// TIA Portal V19 export
FUNCTION_BLOCK "A0304_Navetta_FB"   // FB103, LAD
// stored: MemoryReserve 100, SetENOAutomatically false
   VAR_INPUT
      AreaInterface : "AreaInterface";
      ZSI : "udt_ZoneSafetyInterface";
      DSI_Feed_Testa : "udt_DeviceSafetyInterface";
      DSI_Feed_Coda : "udt_DeviceSafetyInterface";
      DSI_Valve : "udt_DeviceSafetyInterface";
      DataIn : Struct
         OP_Vai_A_Prelievo : Bool;
         OP_Vai_A_Deposito : Bool;
         OP_Prelievo : Bool;
         OP_Deposito : Bool;
         UnloadBenchCaricoMatPres1 : Bool;
         UnloadBenchCaricoMatPres2 : Bool;
         UnloadBenchScaricoMatPres1 : Bool;
         UnloadBenchScaricoMatPres2 : Bool;
         PalettoInternoCoda_LsRest : Bool;
         PalettoInternoCoda_LsWork : Bool;
         PalettoInternoTesta_LsRest : Bool;
         PalettoInternoTesta_LsWork : Bool;
         PalettoEsternoCoda_LsRest : Bool;
         PalettoEsternoCoda_LsWork : Bool;
         PalettoEsternoTesta_LsRest : Bool;
         PalettoEsternoTesta_LsWork : Bool;
      END_STRUCT;
      CIn : Struct
         Manager : Struct
            EnableStopDoorOpeningReq : Bool;
            EnableStopInPhase : Bool;
            EnableStopProgrammed : Bool;
            Control_ON : Bool;
            CanMoveFreely { ExternalAccessible := 'False'; ExternalVisible := 'False'; ExternalWritable := 'False'} : Bool;
            Phase : Struct
               VAI_A_PRELIEVO : Bool;
               PRELIEVO : Bool;
               VAI_A_DEPOSITO : Bool;
               DEPOSITO : Bool;
            END_STRUCT;
         END_STRUCT;
         Sostegno : Struct
            ReadyForDeposito : Bool;
         END_STRUCT;
         Sollevatori : Struct
            Testa : Struct
               InPosDeposito : Bool;
               ActualPos : LReal;
            END_STRUCT;
            Coda : Struct
               InPosDeposito : Bool;
               ActualPos : LReal;
            END_STRUCT;
         END_STRUCT;
         AirOk : Bool;
         CycleModeShortPiece : Bool;
      END_STRUCT;
      Config : Struct
         Navetta : Struct
            Testa : Struct
               Ax : "Positioning_DOL_Machine_Config";
               PalettiEsterni : "ValveMachine_Config";
               PalettiInterni : "ValveMachine_Config";
            END_STRUCT;
            Coda : Struct
               Ax : "Positioning_DOL_Machine_Config";
               PalettiEsterni : "ValveMachine_Config";
               PalettiInterni : "ValveMachine_Config";
            END_STRUCT;
            DelayMissingCondition { ExternalAccessible := 'False'; ExternalVisible := 'False'; ExternalWritable := 'False'} : Time := T#0MS;
         END_STRUCT;
      END_STRUCT;
   END_VAR
   VAR_OUTPUT
      MachineInterface : "MachineInterface";
      COut : Struct
         Testa : Struct
            Ax : "Positioning_DOL_Machine_COut";
            PalettiEsterni : "ValveMachine_COut";
            PalettiInterni : "ValveMachine_COut";
         END_STRUCT;
         Coda : Struct
            Ax : "Positioning_DOL_Machine_COut";
            PalettiEsterni : "ValveMachine_COut";
            PalettiInterni : "ValveMachine_COut";
         END_STRUCT;
         Cumulativo : Struct
            PalettiEsterni : "ValveMachine_COut";
            PalettiInterni : "ValveMachine_COut";
         END_STRUCT;
         ReadyToRecive : Bool;
      END_STRUCT;
      DataOut : Struct
         Testa : Struct
            PalettoEsterno : Struct
               SbloccaggioStelo : Bool;   // 0= Bloccato
               Rest : Bool;
               Work : Bool;
            END_STRUCT;
            PalettoInterno : Struct
               SbloccaggioStelo : Bool;   // 0= Bloccato
               Rest : Bool;
               Work : Bool;
            END_STRUCT;
         END_STRUCT;
         Coda : Struct
            PalettoEsterno : Struct
               SbloccaggioStelo : Bool;
               Rest : Bool;
               Work : Bool;
            END_STRUCT;
            PalettoInterno : Struct
               SbloccaggioStelo : Bool;
               Rest : Bool;
               Work : Bool;
            END_STRUCT;
         END_STRUCT;
      END_STRUCT;
   END_VAR
   VAR_IN_OUT
      Par : Struct
         Ax_Man : "Positioning_DOL_Machine_Par";
         Ax_Testa_Pers : "Positioning_DOL_Machine_Pers_Data";
         Ax_Coda_Pers : "Positioning_DOL_Machine_Pers_Data";
         Enc : Struct
            Testa : "PosFbk_RTN";
            Coda : "PosFbk_RTN";
         END_STRUCT;
      END_STRUCT;
      Par_Mach : Struct
         PosPrePrelievo : LReal;
         PosPrelievo : LReal;
         PosDeposito : LReal;
         ToleranceWindow : LReal;
      END_STRUCT;
   END_VAR
   VAR
      Alarm : Struct
         Testa : Struct
            Ax : "Positioning_DOL_Machine_Alr";
            Enc : "PosFbk_Encoder_Alr";
            PalettiEsterni : "ValveAlr";
            PalettiInterni : "ValveAlr";
         END_STRUCT;
         Coda : Struct
            Ax : "Positioning_DOL_Machine_Alr";
            Enc : "PosFbk_Encoder_Alr";
            PalettiEsterni : "ValveAlr";
            PalettiInterni : "ValveAlr";
         END_STRUCT;
         CheckBothShutMove : Bool;
      END_STRUCT;
      Warning : Struct
         Testa : Struct
            Ax { S7_SetPoint := 'True'} : "Positioning_DOL_Machine_Wng";
            PalettiEsterni : "ValveMachine_Wng";
            PalettiInterni : "ValveMachine_Wng";
         END_STRUCT;
         Coda : Struct
            Ax { S7_SetPoint := 'True'} : "Positioning_DOL_Machine_Wng";
            PalettiEsterni : "ValveMachine_Wng";
            PalettiInterni : "ValveMachine_Wng";
         END_STRUCT;
         MissingCnd : Struct
            OP_VAI_A_PRELIEVO : Bool;   // Mancanza comando arresto
            OP_PRELIEVO : Bool;   // Mancanza consenso lavoro
            OP_VAI_A_DEPOSITO : Bool;   // Mancanza consenso lavoro
            OP_DEPOSITO : Bool;   // Mancanza consenso lavoro
         END_STRUCT;
      END_STRUCT;
      HMI : Struct
         Selection : Struct
            Ax : Int;   // 0= BOTH ; 1= HEAD ; 2= TAIL
            PalettiEsterni : Int;   // 0= BOTH ; 1= HEAD ; 2= TAIL
            PalettiInterni : Int;   // 0= BOTH ; 1= HEAD ; 2= TAIL
         END_STRUCT;
         Testa : Struct
            PbPreset : Bool;
            PresetValue : LReal;
         END_STRUCT;
         Coda : Struct
            PbPreset : Bool;
            PresetValue : LReal;
         END_STRUCT;
      END_STRUCT;
      Sts : Struct
         OP_CanMoveFreely : Bool;
         OP_Vai_A_Prelievo_Cnd : Bool;
         OP_Prelievo_Cnd : Bool;
         OP_Vai_A_Deposito_Cnd : Bool;
         OP_Deposito_Cnd : Bool;
         Coda_PermessoDaSynchOk : Bool;
         Testa_PermessoDaSynchOk : Bool;
         OutOfWorkSpace : Bool;   // Navetta fuori ingombro con impilatore e sollevatore
         GenCndFwd : Bool;
         GenCndBkw : Bool;
         ReloadAirRequest : Bool;
         InPosPrelievo : Bool;
         InPosPrePrelievo : Bool;
         InPosDeposito : Bool;
      END_STRUCT;
      Ctrl : Struct
         Man : Struct
            OP_Vai_A_Prelievo : Bool;
            OP_Prelievo : Bool;
            OP_Vai_A_Deposito : Bool;
            OP_Deposito : Bool;
         END_STRUCT;
         Aut : Struct
            OP_Vai_A_Prelievo : Bool;
            OP_Prelievo : Bool;
            OP_Vai_A_Deposito : Bool;
            OP_Deposito : Bool;
         END_STRUCT;
         OP_Vai_A_Prelievo : Bool;
         OP_Prelievo : Bool;
         OP_Vai_A_Deposito : Bool;
         OP_Deposito : Bool;
         ReloadAir { S7_SetPoint := 'True'} : Bool;
      END_STRUCT;
      Ax_Testa { S7_SetPoint := 'True'} : "Positioning_DOL_Machine_FB";
      Ax_Coda { S7_SetPoint := 'True'} : "Positioning_DOL_Machine_FB";
      PalettiEsterni_Testa { S7_SetPoint := 'True'} : "ValveMachine_FB";
      PalettiEsterni_Coda { S7_SetPoint := 'True'} : "ValveMachine_FB";
      PalettiInterni_Testa { S7_SetPoint := 'True'} : "ValveMachine_FB";
      PalettiInterni_Coda { S7_SetPoint := 'True'} : "ValveMachine_FB";
      BloccaggioStelo_PalettoEsterno_Testa { S7_SetPoint := 'True'} : "Valve";
      BloccaggioStelo_PalettoEsterno_Coda { S7_SetPoint := 'True'} : "Valve";
      Enc_Testa : "PosFbk_SickAFM60";
      Enc_Testa_ITF : "PosFbk_ITF";
      Enc_Coda : "PosFbk_SickAFM60";
      Enc_Coda_ITF : "PosFbk_ITF";
      AUX { ExternalAccessible := 'False'; ExternalVisible := 'False'; ExternalWritable := 'False'} : Struct
         OP_Vai_A_Prelievo : Bool;
         OP_Prelievo : Bool;
         OP_Vai_A_Deposito : Bool;
         OP_Deposito : Bool;
         AirOk : Bool;
         Clock250 : Bool;
      END_STRUCT;
      TON_OP_VAI_A_PRELIEVO_MissingCnd : IEC_TIMER;
      TON_OP_PRELIEVO_MissingCnd : IEC_TIMER;
      TON_OP_VAI_A_DEPOSITO_MissingCnd : IEC_TIMER;
      TON_OP_DEPOSITO_MissingCnd : IEC_TIMER;
      TON_CheckShuttleMove { S7_SetPoint := 'True'} : IEC_TIMER;
      TON_ReloadAir { S7_SetPoint := 'True'} : IEC_TIMER;
      TON_CheckAxis { S7_SetPoint := 'True'} : IEC_TIMER;
      CheckAxisSynch { ExternalAccessible := 'False'; ExternalVisible := 'False'; ExternalWritable := 'False'} : "CheckAxisSynch";
      Sts_PosAxis { S7_SetPoint := 'True'} : Int;
   END_VAR
   VAR_TEMP
      PE : Struct
         OP_Vai_A_Prelievo : Bool;
         OP_Prelievo : Bool;
         OP_Vai_A_Deposito : Bool;
         OP_Deposito : Bool;
         Clock250 : Bool;
      END_STRUCT;
      NE : Struct
         AirOk : Bool;
      END_STRUCT;
      AxTesta_InPosDeposito : Bool;
      AxCoda_InPosDeposito : Bool;
      AxTesta_InPosPrelievo : Bool;
      AxCoda_InPosPrelievo : Bool;
      AxCoda_InPosPrePrelievo : Bool;
      AxTesta_InPosPrePrelievo : Bool;
   END_VAR
   VAR CONSTANT
      "Ax_Fuori Ingombro" : LReal := 800.0;
      MaxDistance : LReal := 5.0;
      MinDistance : LReal := 0.5;
   END_VAR
   // Config.Navetta.Testa.Ax.DelayMissingCondition := T#3S;
   // Config.Navetta.Testa.Ax.CyclicOBTime_ms := 10.0;
   // Config.Navetta.Testa.Ax.Ax.limitMinus := -25.0;
   // Config.Navetta.Testa.Ax.Ax.limitPlus := 2175.0;
   // Config.Navetta.Testa.Ax.Ax.Backlash := 0.0;
   // Config.Navetta.Testa.Ax.Ax.BacklashActivation := FALSE;
   // Config.Navetta.Testa.Ax.Ax.ToleranceWindow := 0.1;
   // Config.Navetta.Testa.Ax.Ax.ToleranceWindowDelay := T#100MS;
   // Config.Navetta.Testa.Ax.Ax.PreCutOff := 0.0;
   // Config.Navetta.Testa.Ax.Ax.PreEndLowSpeed := 0.0;
   // Config.Navetta.Testa.Ax.Ax.PreEndMedSpeed := 0.0;
   // Config.Navetta.Testa.Ax.Ax.ChangeDirectionDelay := T#0MS;
   // Config.Navetta.Testa.Ax.Ax.StandstillVelocity := 0.5;
   // Config.Navetta.Testa.Ax.Ax.StandStillDelay := T#100MS;
   // Config.Navetta.Testa.Ax.Ax.HomingDirection := FALSE;
   // Config.Navetta.Testa.Ax.Ax.RecallTime := 0.0;
   // Config.Navetta.Testa.Ax.Ax.VelocityFilter_T := 10.0;
   // Config.Navetta.Testa.Ax.Ax.VelocityMeasUnit := 2;
   // Config.Navetta.Testa.Ax.Ax.PosFbkDisabled := FALSE;
   // Config.Navetta.Testa.Ax.Ax.FbkCtrlDisabled := TRUE;
   // Config.Navetta.Testa.Ax.Ax_UM2."m" := 1.0;
   // Config.Navetta.Testa.Ax.Ax_UM2.q := 0.0;
   // Config.Navetta.Testa.Ax.S120.SpeedMotor.ReferenceVelocity := 2000.0;
   // Config.Navetta.Testa.Ax.S120.SpeedMotor.InvertDirection := FALSE;
   // Config.Navetta.Testa.Ax.S120.PowerOffDelay := T#5S;
   // Config.Navetta.Testa.Ax.S120.StandstillVelocity := 50.0;
   // Config.Navetta.Testa.Ax.S120.AccTime := 0.25;
   // Config.Navetta.Testa.Ax.S120.DecTime := 0.25;
   // Config.Navetta.Testa.Ax.Fan.Presence := FALSE;
   // Config.Navetta.Testa.Ax.Fan.DelayOff := T#10M;
   // Config.Navetta.Testa.Ax.Brake_Presence := FALSE;
   // Config.Navetta.Testa.PalettiEsterni.DelayPressureRunningTimeout := T#3S;
   // Config.Navetta.Testa.PalettiEsterni.DelayMissingCondition := T#3S;
   // Config.Navetta.Testa.PalettiEsterni.Rest_LsQty := 1;
   // Config.Navetta.Testa.PalettiEsterni.Work_LsQty := 1;
   // Config.Navetta.Testa.PalettiEsterni.Rest_RetainAut := FALSE;
   // Config.Navetta.Testa.PalettiEsterni.Work_RetainAut := FALSE;
   // Config.Navetta.Testa.PalettiEsterni.V.RestLimSwitchExist := TRUE;
   // Config.Navetta.Testa.PalettiEsterni.V.WorkLimSwitchExist := TRUE;
   // Config.Navetta.Testa.PalettiEsterni.V.CheckOilInPressure := FALSE;
   // Config.Navetta.Testa.PalettiEsterni.V.CutRestWhenIsAtRest := TRUE;
   // Config.Navetta.Testa.PalettiEsterni.V.CutWorkWhenIsAtWork := TRUE;
   // Config.Navetta.Testa.PalettiEsterni.V.RestTime := T#0MS;
   // Config.Navetta.Testa.PalettiEsterni.V.WorkTime := T#0MS;
   // Config.Navetta.Testa.PalettiEsterni.V.RestTimeOut := T#6S;
   // Config.Navetta.Testa.PalettiEsterni.V.WorkTimeOut := T#6S;
   // Config.Navetta.Testa.PalettiInterni.DelayPressureRunningTimeout := T#3S;
   // Config.Navetta.Testa.PalettiInterni.DelayMissingCondition := T#3S;
   // Config.Navetta.Testa.PalettiInterni.Rest_LsQty := 1;
   // Config.Navetta.Testa.PalettiInterni.Work_LsQty := 1;
   // Config.Navetta.Testa.PalettiInterni.Rest_RetainAut := FALSE;
   // Config.Navetta.Testa.PalettiInterni.Work_RetainAut := FALSE;
   // Config.Navetta.Testa.PalettiInterni.V.RestLimSwitchExist := TRUE;
   // Config.Navetta.Testa.PalettiInterni.V.WorkLimSwitchExist := TRUE;
   // Config.Navetta.Testa.PalettiInterni.V.CheckOilInPressure := FALSE;
   // Config.Navetta.Testa.PalettiInterni.V.CutRestWhenIsAtRest := TRUE;
   // Config.Navetta.Testa.PalettiInterni.V.CutWorkWhenIsAtWork := TRUE;
   // Config.Navetta.Testa.PalettiInterni.V.RestTime := T#0MS;
   // Config.Navetta.Testa.PalettiInterni.V.WorkTime := T#0MS;
   // Config.Navetta.Testa.PalettiInterni.V.RestTimeOut := T#6S;
   // Config.Navetta.Testa.PalettiInterni.V.WorkTimeOut := T#6S;
   // Config.Navetta.Coda.Ax.DelayMissingCondition := T#3S;
   // Config.Navetta.Coda.Ax.CyclicOBTime_ms := 10.0;
   // Config.Navetta.Coda.Ax.Ax.limitMinus := -25.0;
   // Config.Navetta.Coda.Ax.Ax.limitPlus := 2175.0;
   // Config.Navetta.Coda.Ax.Ax.Backlash := 0.0;
   // Config.Navetta.Coda.Ax.Ax.BacklashActivation := FALSE;
   // Config.Navetta.Coda.Ax.Ax.ToleranceWindow := 0.1;
   // Config.Navetta.Coda.Ax.Ax.ToleranceWindowDelay := T#100MS;
   // Config.Navetta.Coda.Ax.Ax.PreCutOff := 0.0;
   // Config.Navetta.Coda.Ax.Ax.PreEndLowSpeed := 0.0;
   // Config.Navetta.Coda.Ax.Ax.PreEndMedSpeed := 0.0;
   // Config.Navetta.Coda.Ax.Ax.ChangeDirectionDelay := T#0MS;
   // Config.Navetta.Coda.Ax.Ax.StandstillVelocity := 0.5;
   // Config.Navetta.Coda.Ax.Ax.StandStillDelay := T#100MS;
   // Config.Navetta.Coda.Ax.Ax.HomingDirection := FALSE;
   // Config.Navetta.Coda.Ax.Ax.RecallTime := 0.0;
   // Config.Navetta.Coda.Ax.Ax.VelocityFilter_T := 10.0;
   // Config.Navetta.Coda.Ax.Ax.VelocityMeasUnit := 2;
   // Config.Navetta.Coda.Ax.Ax.PosFbkDisabled := FALSE;
   // Config.Navetta.Coda.Ax.Ax.FbkCtrlDisabled := TRUE;
   // Config.Navetta.Coda.Ax.Ax_UM2."m" := 1.0;
   // Config.Navetta.Coda.Ax.Ax_UM2.q := 0.0;
   // Config.Navetta.Coda.Ax.S120.SpeedMotor.ReferenceVelocity := 2200.0;
   // Config.Navetta.Coda.Ax.S120.SpeedMotor.InvertDirection := FALSE;
   // Config.Navetta.Coda.Ax.S120.PowerOffDelay := T#5S;
   // Config.Navetta.Coda.Ax.S120.StandstillVelocity := 50.0;
   // Config.Navetta.Coda.Ax.S120.AccTime := 0.25;
   // Config.Navetta.Coda.Ax.S120.DecTime := 0.25;
   // Config.Navetta.Coda.Ax.Fan.Presence := FALSE;
   // Config.Navetta.Coda.Ax.Fan.DelayOff := T#10M;
   // Config.Navetta.Coda.Ax.Brake_Presence := FALSE;
   // Config.Navetta.Coda.PalettiEsterni.DelayPressureRunningTimeout := T#3S;
   // Config.Navetta.Coda.PalettiEsterni.DelayMissingCondition := T#3S;
   // Config.Navetta.Coda.PalettiEsterni.Rest_LsQty := 1;
   // Config.Navetta.Coda.PalettiEsterni.Work_LsQty := 1;
   // Config.Navetta.Coda.PalettiEsterni.Rest_RetainAut := FALSE;
   // Config.Navetta.Coda.PalettiEsterni.Work_RetainAut := FALSE;
   // Config.Navetta.Coda.PalettiEsterni.V.RestLimSwitchExist := TRUE;
   // Config.Navetta.Coda.PalettiEsterni.V.WorkLimSwitchExist := TRUE;
   // Config.Navetta.Coda.PalettiEsterni.V.CheckOilInPressure := FALSE;
   // Config.Navetta.Coda.PalettiEsterni.V.CutRestWhenIsAtRest := TRUE;
   // Config.Navetta.Coda.PalettiEsterni.V.CutWorkWhenIsAtWork := TRUE;
   // Config.Navetta.Coda.PalettiEsterni.V.RestTime := T#0MS;
   // Config.Navetta.Coda.PalettiEsterni.V.WorkTime := T#0MS;
   // Config.Navetta.Coda.PalettiEsterni.V.RestTimeOut := T#6S;
   // Config.Navetta.Coda.PalettiEsterni.V.WorkTimeOut := T#6S;
   // Config.Navetta.Coda.PalettiInterni.DelayPressureRunningTimeout := T#3S;
   // Config.Navetta.Coda.PalettiInterni.DelayMissingCondition := T#3S;
   // Config.Navetta.Coda.PalettiInterni.Rest_LsQty := 1;
   // Config.Navetta.Coda.PalettiInterni.Work_LsQty := 1;
   // Config.Navetta.Coda.PalettiInterni.Rest_RetainAut := FALSE;
   // Config.Navetta.Coda.PalettiInterni.Work_RetainAut := FALSE;
   // Config.Navetta.Coda.PalettiInterni.V.RestLimSwitchExist := TRUE;
   // Config.Navetta.Coda.PalettiInterni.V.WorkLimSwitchExist := TRUE;
   // Config.Navetta.Coda.PalettiInterni.V.CheckOilInPressure := FALSE;
   // Config.Navetta.Coda.PalettiInterni.V.CutRestWhenIsAtRest := TRUE;
   // Config.Navetta.Coda.PalettiInterni.V.CutWorkWhenIsAtWork := TRUE;
   // Config.Navetta.Coda.PalettiInterni.V.RestTime := T#0MS;
   // Config.Navetta.Coda.PalettiInterni.V.WorkTime := T#0MS;
   // Config.Navetta.Coda.PalettiInterni.V.RestTimeOut := T#6S;
   // Config.Navetta.Coda.PalettiInterni.V.WorkTimeOut := T#6S;
   VAR_TEMP   // added for the SCL form of the ladder/FBD networks
      _w1 : Bool;
      _w2 : Bool;
      _w3 : Bool;
      _w4 : Bool;
   END_VAR
BEGIN

REGION Network 1 (SCL): Reset allarmi
   IF #AreaInterface.RstAlarms THEN
       #Alarm.CheckBothShutMove := FALSE;
   END_IF;
END_REGION

REGION Network 2: <+>
END_REGION

REGION Network 3: <<<<<<<<<<<<<<<<<<< OPERAZIONI >>>>>>>>>>>>>>>>>>>>>>>>
END_REGION

REGION Network 4: Operazione può muoversi liberamente perchè non sposta nessun BEAM
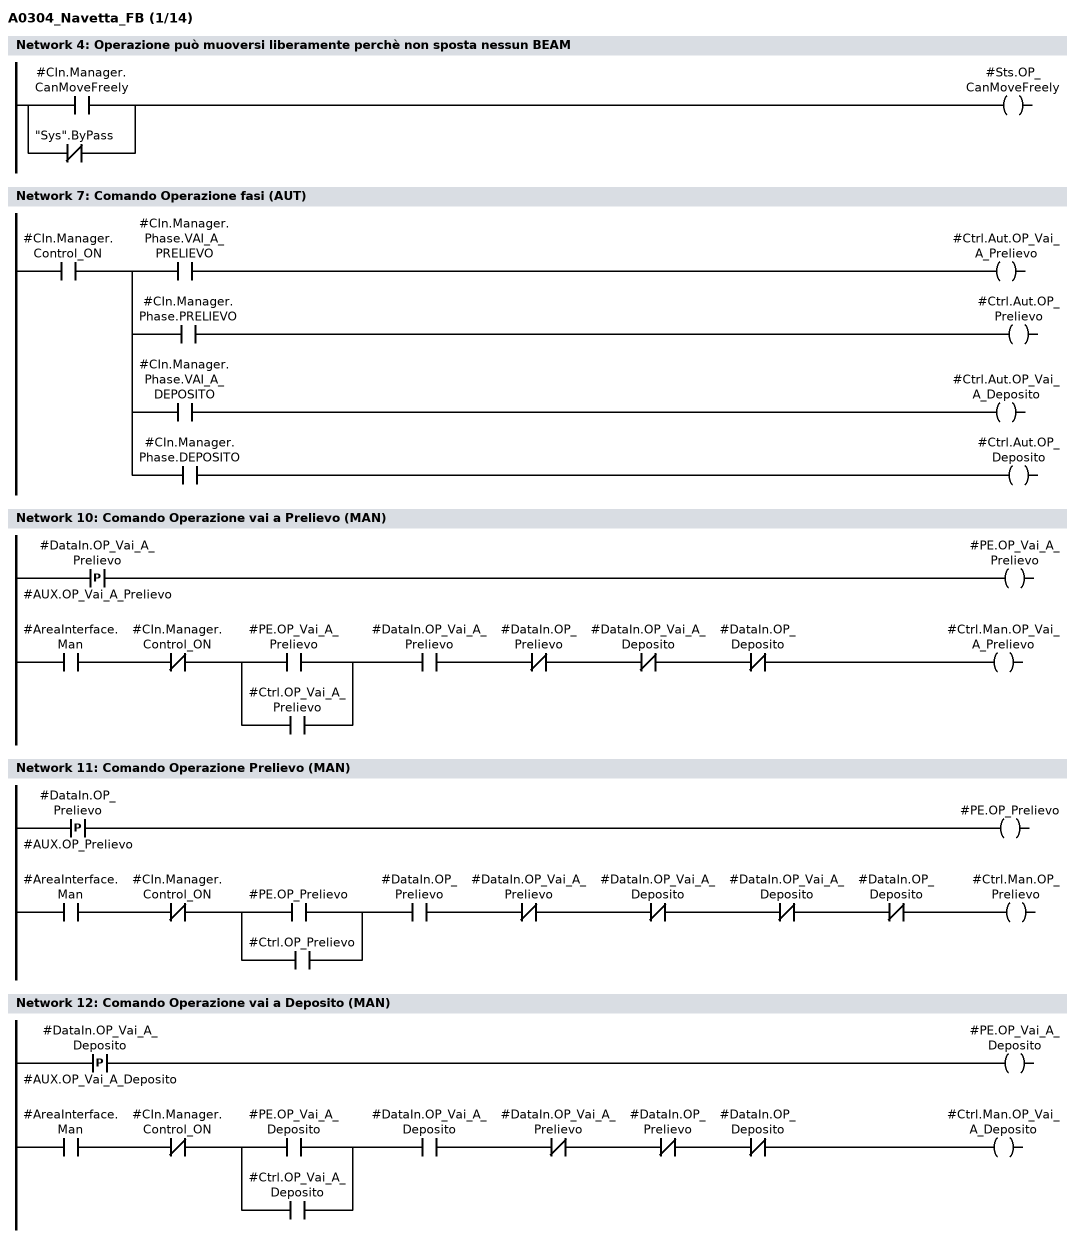
   RUNG wire#powerrail
      Contact( #CIn.Manager.CanMoveFreely )
      wire#w1
      Coil( #Sts.OP_CanMoveFreely )
   END_RUNG
   RUNG wire#powerrail
      I_Contact( "Sys".ByPass )
   END_RUNG wire#w1
   // the same network as SCL:
   #Sts.OP_CanMoveFreely := #CIn.Manager.CanMoveFreely OR NOT "Sys".ByPass;
END_REGION

REGION Network 5: <+>
END_REGION

REGION Network 6: < OPERAZIONI AUTOMATICO >
END_REGION

REGION Network 7: Comando Operazione fasi (AUT)
   RUNG wire#powerrail
      Contact( #CIn.Manager.Control_ON )
      wire#w1
      Contact( #CIn.Manager.Phase.VAI_A_PRELIEVO )
      Coil( #Ctrl.Aut.OP_Vai_A_Prelievo )
   END_RUNG
   RUNG wire#w1
      Contact( #CIn.Manager.Phase.PRELIEVO )
      Coil( #Ctrl.Aut.OP_Prelievo )
   END_RUNG
   RUNG wire#w1
      Contact( #CIn.Manager.Phase.VAI_A_DEPOSITO )
      Coil( #Ctrl.Aut.OP_Vai_A_Deposito )
   END_RUNG
   RUNG wire#w1
      Contact( #CIn.Manager.Phase.DEPOSITO )
      Coil( #Ctrl.Aut.OP_Deposito )
   END_RUNG
   // the same network as SCL:
   #Ctrl.Aut.OP_Vai_A_Prelievo := #CIn.Manager.Control_ON AND #CIn.Manager.Phase.VAI_A_PRELIEVO;
   #Ctrl.Aut.OP_Prelievo := #CIn.Manager.Control_ON AND #CIn.Manager.Phase.PRELIEVO;
   #Ctrl.Aut.OP_Vai_A_Deposito := #CIn.Manager.Control_ON AND #CIn.Manager.Phase.VAI_A_DEPOSITO;
   #Ctrl.Aut.OP_Deposito := #CIn.Manager.Control_ON AND #CIn.Manager.Phase.DEPOSITO;
END_REGION

REGION Network 8: <+>
END_REGION

REGION Network 9: < OPERAZIONI MANUALI >
END_REGION

REGION Network 10: Comando Operazione vai a Prelievo (MAN)
   RUNG wire#powerrail
      P_Contact(operand := #DataIn.OP_Vai_A_Prelievo, bit := #AUX.OP_Vai_A_Prelievo)
      Coil( #PE.OP_Vai_A_Prelievo )
   END_RUNG
   RUNG wire#powerrail
      Contact( #AreaInterface.Man )
      I_Contact( #CIn.Manager.Control_ON )
      wire#w1
      Contact( #PE.OP_Vai_A_Prelievo )
      wire#w2
      Contact( #DataIn.OP_Vai_A_Prelievo )
      I_Contact( #DataIn.OP_Prelievo )
      I_Contact( #DataIn.OP_Vai_A_Deposito )
      I_Contact( #DataIn.OP_Deposito )
      Coil( #Ctrl.Man.OP_Vai_A_Prelievo )
   END_RUNG
   RUNG wire#w1
      Contact( #Ctrl.OP_Vai_A_Prelievo )
   END_RUNG wire#w2
   // the same network as SCL:
   #_w1 := #DataIn.OP_Vai_A_Prelievo AND NOT #AUX.OP_Vai_A_Prelievo;   // rising edge of #DataIn.OP_Vai_A_Prelievo
   #AUX.OP_Vai_A_Prelievo := #DataIn.OP_Vai_A_Prelievo;
   #PE.OP_Vai_A_Prelievo := #_w1;
   #Ctrl.Man.OP_Vai_A_Prelievo := #AreaInterface.Man AND NOT #CIn.Manager.Control_ON AND (#PE.OP_Vai_A_Prelievo OR #Ctrl.OP_Vai_A_Prelievo) AND #DataIn.OP_Vai_A_Prelievo AND NOT #DataIn.OP_Prelievo AND NOT #DataIn.OP_Vai_A_Deposito AND NOT #DataIn.OP_Deposito;
END_REGION

REGION Network 11: Comando Operazione Prelievo (MAN)
   RUNG wire#powerrail
      P_Contact(operand := #DataIn.OP_Prelievo, bit := #AUX.OP_Prelievo)
      Coil( #PE.OP_Prelievo )
   END_RUNG
   RUNG wire#powerrail
      Contact( #AreaInterface.Man )
      I_Contact( #CIn.Manager.Control_ON )
      wire#w1
      Contact( #PE.OP_Prelievo )
      wire#w2
      Contact( #DataIn.OP_Prelievo )
      I_Contact( #DataIn.OP_Vai_A_Prelievo )
      I_Contact( #DataIn.OP_Vai_A_Deposito )
      I_Contact( #DataIn.OP_Vai_A_Deposito )
      I_Contact( #DataIn.OP_Deposito )
      Coil( #Ctrl.Man.OP_Prelievo )
   END_RUNG
   RUNG wire#w1
      Contact( #Ctrl.OP_Prelievo )
   END_RUNG wire#w2
   // the same network as SCL:
   #_w1 := #DataIn.OP_Prelievo AND NOT #AUX.OP_Prelievo;   // rising edge of #DataIn.OP_Prelievo
   #AUX.OP_Prelievo := #DataIn.OP_Prelievo;
   #PE.OP_Prelievo := #_w1;
   #Ctrl.Man.OP_Prelievo := #AreaInterface.Man AND NOT #CIn.Manager.Control_ON AND (#PE.OP_Prelievo OR #Ctrl.OP_Prelievo) AND #DataIn.OP_Prelievo AND NOT #DataIn.OP_Vai_A_Prelievo AND NOT #DataIn.OP_Vai_A_Deposito AND NOT #DataIn.OP_Vai_A_Deposito AND NOT #DataIn.OP_Deposito;
END_REGION

REGION Network 12: Comando Operazione vai a Deposito (MAN)
   RUNG wire#powerrail
      P_Contact(operand := #DataIn.OP_Vai_A_Deposito, bit := #AUX.OP_Vai_A_Deposito)
      Coil( #PE.OP_Vai_A_Deposito )
   END_RUNG
   RUNG wire#powerrail
      Contact( #AreaInterface.Man )
      I_Contact( #CIn.Manager.Control_ON )
      wire#w1
      Contact( #PE.OP_Vai_A_Deposito )
      wire#w2
      Contact( #DataIn.OP_Vai_A_Deposito )
      I_Contact( #DataIn.OP_Vai_A_Prelievo )
      I_Contact( #DataIn.OP_Prelievo )
      I_Contact( #DataIn.OP_Deposito )
      Coil( #Ctrl.Man.OP_Vai_A_Deposito )
   END_RUNG
   RUNG wire#w1
      Contact( #Ctrl.OP_Vai_A_Deposito )
   END_RUNG wire#w2
   // the same network as SCL:
   #_w1 := #DataIn.OP_Vai_A_Deposito AND NOT #AUX.OP_Vai_A_Deposito;   // rising edge of #DataIn.OP_Vai_A_Deposito
   #AUX.OP_Vai_A_Deposito := #DataIn.OP_Vai_A_Deposito;
   #PE.OP_Vai_A_Deposito := #_w1;
   #Ctrl.Man.OP_Vai_A_Deposito := #AreaInterface.Man AND NOT #CIn.Manager.Control_ON AND (#PE.OP_Vai_A_Deposito OR #Ctrl.OP_Vai_A_Deposito) AND #DataIn.OP_Vai_A_Deposito AND NOT #DataIn.OP_Vai_A_Prelievo AND NOT #DataIn.OP_Prelievo AND NOT #DataIn.OP_Deposito;
END_REGION

REGION Network 13: Comando Operazione Deposito (MAN)
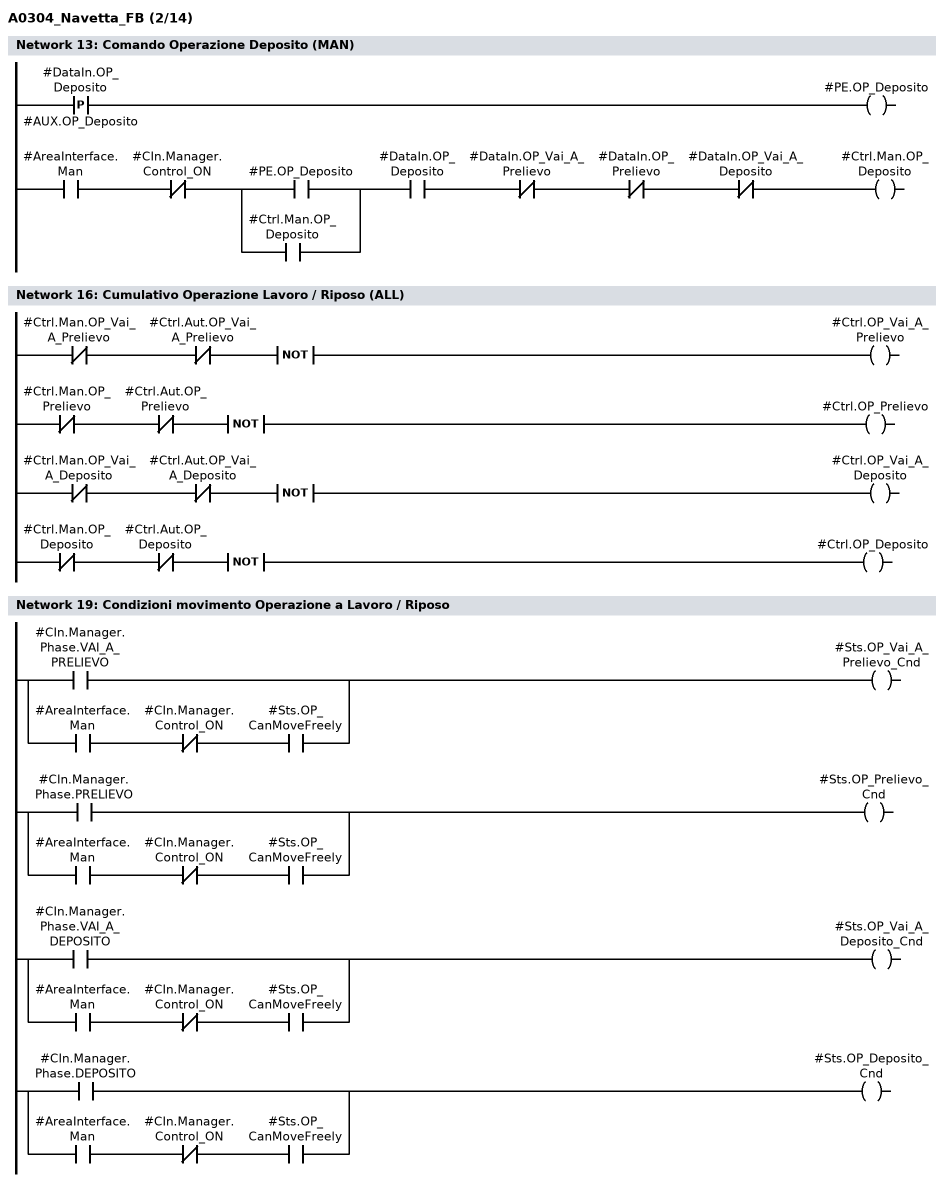
   RUNG wire#powerrail
      P_Contact(operand := #DataIn.OP_Deposito, bit := #AUX.OP_Deposito)
      Coil( #PE.OP_Deposito )
   END_RUNG
   RUNG wire#powerrail
      Contact( #AreaInterface.Man )
      I_Contact( #CIn.Manager.Control_ON )
      wire#w1
      Contact( #PE.OP_Deposito )
      wire#w2
      Contact( #DataIn.OP_Deposito )
      I_Contact( #DataIn.OP_Vai_A_Prelievo )
      I_Contact( #DataIn.OP_Prelievo )
      I_Contact( #DataIn.OP_Vai_A_Deposito )
      Coil( #Ctrl.Man.OP_Deposito )
   END_RUNG
   RUNG wire#w1
      Contact( #Ctrl.Man.OP_Deposito )
   END_RUNG wire#w2
   // the same network as SCL:
   #_w1 := #DataIn.OP_Deposito AND NOT #AUX.OP_Deposito;   // rising edge of #DataIn.OP_Deposito
   #AUX.OP_Deposito := #DataIn.OP_Deposito;
   #PE.OP_Deposito := #_w1;
   #Ctrl.Man.OP_Deposito := #AreaInterface.Man AND NOT #CIn.Manager.Control_ON AND (#PE.OP_Deposito OR #Ctrl.Man.OP_Deposito) AND #DataIn.OP_Deposito AND NOT #DataIn.OP_Vai_A_Prelievo AND NOT #DataIn.OP_Prelievo AND NOT #DataIn.OP_Vai_A_Deposito;
END_REGION

REGION Network 14: <+>
END_REGION

REGION Network 15: < CUMULATIVO OPERAZIONI >
END_REGION

REGION Network 16: Cumulativo Operazione Lavoro / Riposo (ALL)
   RUNG wire#powerrail
      I_Contact( #Ctrl.Man.OP_Vai_A_Prelievo )
      I_Contact( #Ctrl.Aut.OP_Vai_A_Prelievo )
      Not()
      Coil( #Ctrl.OP_Vai_A_Prelievo )
   END_RUNG
   RUNG wire#powerrail
      I_Contact( #Ctrl.Man.OP_Prelievo )
      I_Contact( #Ctrl.Aut.OP_Prelievo )
      Not()
      Coil( #Ctrl.OP_Prelievo )
   END_RUNG
   RUNG wire#powerrail
      I_Contact( #Ctrl.Man.OP_Vai_A_Deposito )
      I_Contact( #Ctrl.Aut.OP_Vai_A_Deposito )
      Not()
      Coil( #Ctrl.OP_Vai_A_Deposito )
   END_RUNG
   RUNG wire#powerrail
      I_Contact( #Ctrl.Man.OP_Deposito )
      I_Contact( #Ctrl.Aut.OP_Deposito )
      Not()
      Coil( #Ctrl.OP_Deposito )
   END_RUNG
   // the same network as SCL:
   #Ctrl.OP_Vai_A_Prelievo := NOT (NOT #Ctrl.Man.OP_Vai_A_Prelievo AND NOT #Ctrl.Aut.OP_Vai_A_Prelievo);
   #Ctrl.OP_Prelievo := NOT (NOT #Ctrl.Man.OP_Prelievo AND NOT #Ctrl.Aut.OP_Prelievo);
   #Ctrl.OP_Vai_A_Deposito := NOT (NOT #Ctrl.Man.OP_Vai_A_Deposito AND NOT #Ctrl.Aut.OP_Vai_A_Deposito);
   #Ctrl.OP_Deposito := NOT (NOT #Ctrl.Man.OP_Deposito AND NOT #Ctrl.Aut.OP_Deposito);
END_REGION

REGION Network 17: <+>
END_REGION

REGION Network 18: < CONDIZIONI MOVIMENTO >
END_REGION

REGION Network 19: Condizioni movimento Operazione a Lavoro / Riposo
   RUNG wire#powerrail
      Contact( #CIn.Manager.Phase.VAI_A_PRELIEVO )
      wire#w1
      Coil( #Sts.OP_Vai_A_Prelievo_Cnd )
   END_RUNG
   RUNG wire#powerrail
      Contact( #AreaInterface.Man )
      I_Contact( #CIn.Manager.Control_ON )
      Contact( #Sts.OP_CanMoveFreely )
   END_RUNG wire#w1
   RUNG wire#powerrail
      Contact( #CIn.Manager.Phase.PRELIEVO )
      wire#w2
      Coil( #Sts.OP_Prelievo_Cnd )
   END_RUNG
   RUNG wire#powerrail
      Contact( #AreaInterface.Man )
      I_Contact( #CIn.Manager.Control_ON )
      Contact( #Sts.OP_CanMoveFreely )
   END_RUNG wire#w2
   RUNG wire#powerrail
      Contact( #CIn.Manager.Phase.VAI_A_DEPOSITO )
      wire#w3
      Coil( #Sts.OP_Vai_A_Deposito_Cnd )
   END_RUNG
   RUNG wire#powerrail
      Contact( #AreaInterface.Man )
      I_Contact( #CIn.Manager.Control_ON )
      Contact( #Sts.OP_CanMoveFreely )
   END_RUNG wire#w3
   RUNG wire#powerrail
      Contact( #CIn.Manager.Phase.DEPOSITO )
      wire#w4
      Coil( #Sts.OP_Deposito_Cnd )
   END_RUNG
   RUNG wire#powerrail
      Contact( #AreaInterface.Man )
      I_Contact( #CIn.Manager.Control_ON )
      Contact( #Sts.OP_CanMoveFreely )
   END_RUNG wire#w4
   // the same network as SCL:
   #Sts.OP_Vai_A_Prelievo_Cnd := #CIn.Manager.Phase.VAI_A_PRELIEVO OR (#AreaInterface.Man AND NOT #CIn.Manager.Control_ON AND #Sts.OP_CanMoveFreely);
   #Sts.OP_Prelievo_Cnd := #CIn.Manager.Phase.PRELIEVO OR (#AreaInterface.Man AND NOT #CIn.Manager.Control_ON AND #Sts.OP_CanMoveFreely);
   #Sts.OP_Vai_A_Deposito_Cnd := #CIn.Manager.Phase.VAI_A_DEPOSITO OR (#AreaInterface.Man AND NOT #CIn.Manager.Control_ON AND #Sts.OP_CanMoveFreely);
   #Sts.OP_Deposito_Cnd := #CIn.Manager.Phase.DEPOSITO OR (#AreaInterface.Man AND NOT #CIn.Manager.Control_ON AND #Sts.OP_CanMoveFreely);
END_REGION

REGION Network 20: <+>
END_REGION

REGION Network 21: <+>
END_REGION

REGION Network 22: <<<<<<<<<<<<<<<<<<< SEQUENZA COMANDI >>>>>>>>>>>>>>>>>>>>>>>>
END_REGION

REGION Network 23: Ax Navetta in posizione
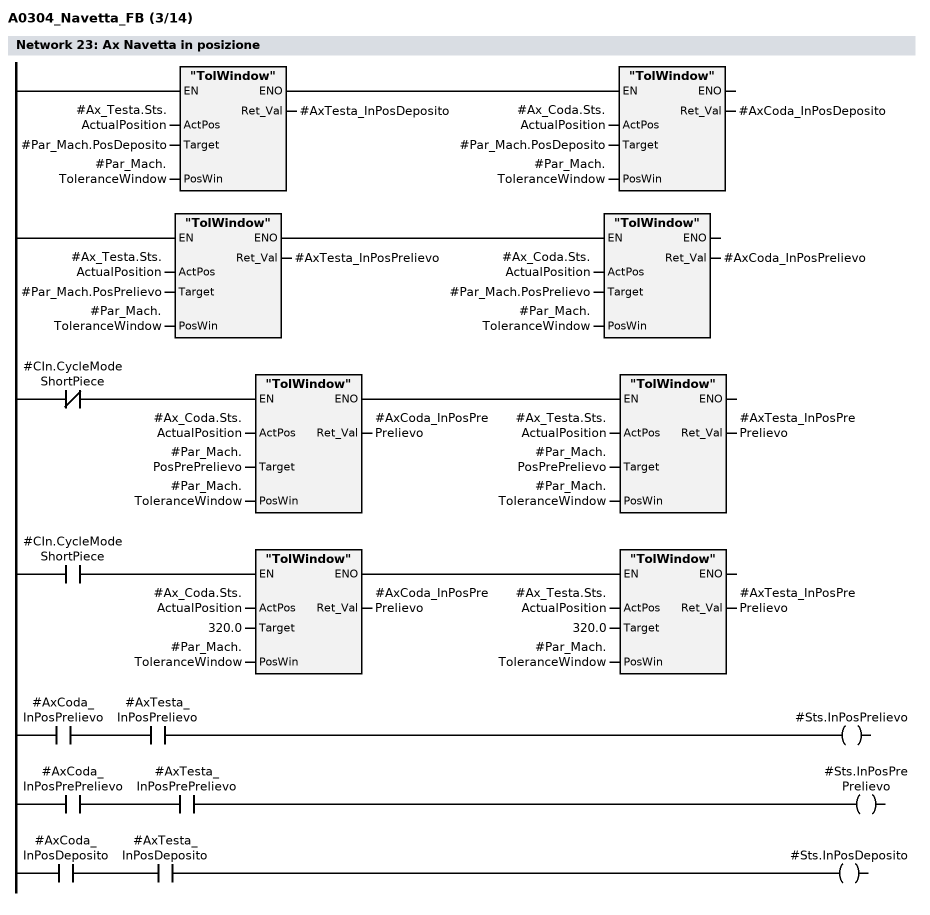
   RUNG wire#powerrail
      "TolWindow"(ActPos := #Ax_Testa.Sts.ActualPosition, Target := #Par_Mach.PosDeposito, PosWin := #Par_Mach.ToleranceWindow, Ret_Val => #AxTesta_InPosDeposito)
      "TolWindow"(ActPos := #Ax_Coda.Sts.ActualPosition, Target := #Par_Mach.PosDeposito, PosWin := #Par_Mach.ToleranceWindow, Ret_Val => #AxCoda_InPosDeposito)
   END_RUNG
   RUNG wire#powerrail
      "TolWindow"(ActPos := #Ax_Testa.Sts.ActualPosition, Target := #Par_Mach.PosPrelievo, PosWin := #Par_Mach.ToleranceWindow, Ret_Val => #AxTesta_InPosPrelievo)
      "TolWindow"(ActPos := #Ax_Coda.Sts.ActualPosition, Target := #Par_Mach.PosPrelievo, PosWin := #Par_Mach.ToleranceWindow, Ret_Val => #AxCoda_InPosPrelievo)
   END_RUNG
   RUNG wire#powerrail
      I_Contact( #CIn.CycleModeShortPiece )
      "TolWindow"(ActPos := #Ax_Coda.Sts.ActualPosition, Target := #Par_Mach.PosPrePrelievo, PosWin := #Par_Mach.ToleranceWindow, Ret_Val => #AxCoda_InPosPrePrelievo)
      "TolWindow"(ActPos := #Ax_Testa.Sts.ActualPosition, Target := #Par_Mach.PosPrePrelievo, PosWin := #Par_Mach.ToleranceWindow, Ret_Val => #AxTesta_InPosPrePrelievo)
   END_RUNG
   RUNG wire#powerrail
      Contact( #CIn.CycleModeShortPiece )
      "TolWindow"(ActPos := #Ax_Coda.Sts.ActualPosition, Target := 320.0, PosWin := #Par_Mach.ToleranceWindow, Ret_Val => #AxCoda_InPosPrePrelievo)
      "TolWindow"(ActPos := #Ax_Testa.Sts.ActualPosition, Target := 320.0, PosWin := #Par_Mach.ToleranceWindow, Ret_Val => #AxTesta_InPosPrePrelievo)
   END_RUNG
   RUNG wire#powerrail
      Contact( #AxCoda_InPosPrelievo )
      Contact( #AxTesta_InPosPrelievo )
      Coil( #Sts.InPosPrelievo )
   END_RUNG
   RUNG wire#powerrail
      Contact( #AxCoda_InPosPrePrelievo )
      Contact( #AxTesta_InPosPrePrelievo )
      Coil( #Sts.InPosPrePrelievo )
   END_RUNG
   RUNG wire#powerrail
      Contact( #AxCoda_InPosDeposito )
      Contact( #AxTesta_InPosDeposito )
      Coil( #Sts.InPosDeposito )
   END_RUNG
   // the same network as SCL:
   #AxTesta_InPosDeposito := "TolWindow"(ActPos := #Ax_Testa.Sts.ActualPosition,
                           Target := #Par_Mach.PosDeposito,
                           PosWin := #Par_Mach.ToleranceWindow,
                           ENO => #_w1);
   IF #_w1 THEN
       #AxCoda_InPosDeposito := "TolWindow"(ActPos := #Ax_Coda.Sts.ActualPosition,
                               Target := #Par_Mach.PosDeposito,
                               PosWin := #Par_Mach.ToleranceWindow);
   END_IF;
   #AxTesta_InPosPrelievo := "TolWindow"(ActPos := #Ax_Testa.Sts.ActualPosition,
                           Target := #Par_Mach.PosPrelievo,
                           PosWin := #Par_Mach.ToleranceWindow,
                           ENO => #_w2);
   IF #_w2 THEN
       #AxCoda_InPosPrelievo := "TolWindow"(ActPos := #Ax_Coda.Sts.ActualPosition,
                               Target := #Par_Mach.PosPrelievo,
                               PosWin := #Par_Mach.ToleranceWindow);
   END_IF;
   #AxCoda_InPosPrePrelievo := "TolWindow"(EN := NOT #CIn.CycleModeShortPiece,
                           ActPos := #Ax_Coda.Sts.ActualPosition,
                           Target := #Par_Mach.PosPrePrelievo,
                           PosWin := #Par_Mach.ToleranceWindow,
                           ENO => #_w3);
   IF #_w3 THEN
       #AxTesta_InPosPrePrelievo := "TolWindow"(ActPos := #Ax_Testa.Sts.ActualPosition,
                               Target := #Par_Mach.PosPrePrelievo,
                               PosWin := #Par_Mach.ToleranceWindow);
   END_IF;
   #AxCoda_InPosPrePrelievo := "TolWindow"(EN := #CIn.CycleModeShortPiece,
                           ActPos := #Ax_Coda.Sts.ActualPosition,
                           Target := 320.0,
                           PosWin := #Par_Mach.ToleranceWindow,
                           ENO => #_w4);
   IF #_w4 THEN
       #AxTesta_InPosPrePrelievo := "TolWindow"(ActPos := #Ax_Testa.Sts.ActualPosition,
                               Target := 320.0,
                               PosWin := #Par_Mach.ToleranceWindow);
   END_IF;
   #Sts.InPosPrelievo := #AxCoda_InPosPrelievo AND #AxTesta_InPosPrelievo;
   #Sts.InPosPrePrelievo := #AxCoda_InPosPrePrelievo AND #AxTesta_InPosPrePrelievo;
   #Sts.InPosDeposito := #AxCoda_InPosDeposito AND #AxTesta_InPosDeposito;
END_REGION

REGION Network 24 (SCL): Sincronizzazione tra asse testa e asse coda
   #CheckAxisSynch(Ax1_Pos:=#Ax_Testa.Sts.ActualPosition,
                   Ax2_Pos:=#Ax_Coda.Sts.ActualPosition,
                   TargetPos:=#Ax_Testa.Ctrl.Pos,
                   MaxDistance:=#MaxDistance,
                   MinDistance:=#MinDistance,
                   Ax1_SynchOk=> #Sts.Testa_PermessoDaSynchOk,
                   Ax2_SynchOk=> #Sts.Coda_PermessoDaSynchOk);
END_REGION

REGION Network 25: <+>
END_REGION

REGION Network 26 (SCL): CIn Abilitazioni Manager
   //Stop Door Opening Request
   #Ax_Testa.CIn.Manager.EnableStopDoorOpeningReq := #Ax_Coda.CIn.Manager.EnableStopDoorOpeningReq :=
   #PalettiEsterni_Testa.Cin.Manager.EnableStopDoorOpeningReq := #PalettiEsterni_Coda.Cin.Manager.EnableStopDoorOpeningReq :=
   #PalettiInterni_Testa.Cin.Manager.EnableStopDoorOpeningReq := #PalettiInterni_Coda.Cin.Manager.EnableStopDoorOpeningReq := #CIn.Manager.EnableStopDoorOpeningReq;

   //Stop In Phase
   #Ax_Testa.CIn.Manager.EnableStopInPhase := #Ax_Coda.CIn.Manager.EnableStopInPhase :=
   #PalettiEsterni_Testa.Cin.Manager.EnableStopInPhase := #PalettiEsterni_Coda.Cin.Manager.EnableStopInPhase :=
   #PalettiInterni_Testa.Cin.Manager.EnableStopInPhase := #PalettiInterni_Coda.Cin.Manager.EnableStopInPhase := #CIn.Manager.EnableStopInPhase;

   //Stop Programmed
   #Ax_Testa.CIn.Manager.EnableStopProgrammed := #Ax_Coda.CIn.Manager.EnableStopProgrammed :=
   #PalettiEsterni_Testa.Cin.Manager.EnableStopProgrammed := #PalettiEsterni_Coda.Cin.Manager.EnableStopProgrammed :=
   #PalettiInterni_Testa.Cin.Manager.EnableStopProgrammed := #PalettiInterni_Coda.Cin.Manager.EnableStopProgrammed := #CIn.Manager.EnableStopProgrammed;
END_REGION

REGION Network 27 (SCL): Cin Manager (Esecuzione sequenza comandi)
   //CTRL ON
   #Ax_Testa.CIn.Manager.Control_ON := #Ax_Coda.CIn.Manager.Control_ON :=
   #PalettiEsterni_Testa.Cin.Manager.Control_ON := #PalettiEsterni_Coda.Cin.Manager.Control_ON :=
   #PalettiInterni_Testa.Cin.Manager.Control_ON := #PalettiInterni_Coda.Cin.Manager.Control_ON := #Ctrl.OP_Prelievo OR #Ctrl.OP_Vai_A_Deposito OR #Ctrl.OP_Vai_A_Prelievo OR  #Ctrl.OP_Deposito;

   #Ax_Testa.CIn.Manager.Speed := #Ax_Coda.CIn.Manager.Speed :=100;

   #TON_CheckAxis.TON(IN := #Sts_PosAxis = 2 OR #Sts_PosAxis = 3,
                      PT := T#1S);


   //Power On Assi
   #Ax_Coda.CIn.ExternalPowerOn := #Ax_Testa.CIn.ExternalPowerOn := #Ctrl.OP_Vai_A_Prelievo OR #Ctrl.OP_Vai_A_Deposito OR #Ctrl.OP_Prelievo;

   IF #Sts_PosAxis = 3 AND  ABS(#Ax_Testa.Sts.ActualPosition - #Ax_Coda.Sts.ActualPosition) > #MaxDistance THEN
       #Sts_PosAxis := 0;
   END_IF;

   IF NOT #Ctrl.OP_Vai_A_Deposito AND NOT #Ctrl.OP_Vai_A_Prelievo AND NOT #Ctrl.OP_Prelievo THEN
       #Sts_PosAxis := 0;
   END_IF;

   IF #Sts_PosAxis = 0 THEN

       #Ax_Testa.CIn.Manager.MoveToPos := #Ax_Coda.CIn.Manager.MoveToPos := FALSE;

       IF #Ctrl.OP_Vai_A_Deposito OR #Ctrl.OP_Vai_A_Prelievo OR #Ctrl.OP_Prelievo THEN
           IF ABS(#Ax_Testa.Sts.ActualPosition - #Ax_Coda.Sts.ActualPosition) > #MaxDistance THEN

               #Ax_Testa.CIn.Manager.Pos := #Ax_Coda.Sts.ActualPosition;
               #Ax_Coda.CIn.Manager.Pos := #Ax_Coda.Sts.ActualPosition;
               #Ax_Coda.CIn.Manager.MoveToPos := TRUE;
               #Ax_Testa.CIn.Manager.MoveToPos := TRUE;


               #Sts_PosAxis := 1;
           ELSE
               #Sts_PosAxis := 3;
           END_IF;

       END_IF;
   END_IF;

   IF #Sts_PosAxis = 1 THEN

       IF ABS(#Ax_Testa.Sts.ActualPosition - #Ax_Coda.Sts.ActualPosition) <#MinDistance THEN
           #Ax_Testa.CIn.Manager.MoveToPos := FALSE;
           #Ax_Coda.CIn.Manager.MoveToPos := FALSE;

           #Sts_PosAxis := 2;

       END_IF;

   END_IF;

   IF #Sts_PosAxis = 2 THEN


           #Ax_Testa.CIn.Manager.MoveToPos := FALSE;
           #Ax_Coda.CIn.Manager.MoveToPos := FALSE;

           IF #Ax_Coda.COut.Standstill AND #Ax_Testa.COut.Standstill AND #TON_CheckAxis.Q THEN

               #Sts_PosAxis := 3;
           END_IF;

   END_IF;

   IF #Sts_PosAxis = 3 AND NOT #Alarm.CheckBothShutMove THEN

       #Ax_Testa.CIn.Manager.MoveToPos := FALSE;
       #Ax_Coda.CIn.Manager.MoveToPos := FALSE;


       IF #Ctrl.OP_Vai_A_Prelievo AND #Sts.OP_Vai_A_Prelievo_Cnd THEN

           #Ax_Testa.CIn.Manager.Speed := #Ax_Coda.CIn.Manager.Speed := 100;

           // Paletti Interni
           #PalettiInterni_Testa.Cin.Manager.Rest := NOT #PalettiInterni_Testa.COut.Rest;
           #PalettiInterni_Coda.Cin.Manager.Rest := NOT #PalettiInterni_Coda.COut.Rest;

           // Paletti Esterni
           #PalettiEsterni_Testa.Cin.Manager.Rest := NOT #PalettiEsterni_Testa.COut.Rest;
           #PalettiEsterni_Coda.Cin.Manager.Rest := NOT #PalettiEsterni_Coda.COut.Rest;

           // Trasporto in posizione di Prelievo
           IF NOT #CIn.CycleModeShortPiece THEN
               #Ax_Coda.CIn.Manager.Pos := #Ax_Testa.CIn.Manager.Pos := #Par_Mach.PosPrePrelievo;
           ELSE
               #Ax_Coda.CIn.Manager.Pos := #Ax_Testa.CIn.Manager.Pos := 320;
           END_IF;


           #Ax_Testa.CIn.Manager.MoveToPos := NOT #AxTesta_InPosPrePrelievo AND #PalettiInterni_Testa.COut.Rest AND #PalettiInterni_Coda.COut.Rest
           AND #PalettiEsterni_Testa.COut.Rest AND #PalettiEsterni_Coda.COut.Rest AND #Ax_Testa.S120.Sts.AxisEnabled AND #Ax_Coda.S120.Sts.AxisEnabled AND #TON_CheckAxis.Q;


           #Ax_Coda.CIn.Manager.MoveToPos := NOT #AxCoda_InPosPrePrelievo AND #PalettiInterni_Testa.COut.Rest AND #PalettiInterni_Coda.COut.Rest
           AND #PalettiEsterni_Testa.COut.Rest AND #PalettiEsterni_Coda.COut.Rest AND #Ax_Testa.S120.Sts.AxisEnabled AND #Ax_Coda.S120.Sts.AxisEnabled AND #TON_CheckAxis.Q;




       ELSIF #Ctrl.OP_Vai_A_Deposito AND #Sts.OP_Vai_A_Deposito_Cnd THEN

           #Ax_Testa.CIn.Manager.Speed := #Ax_Coda.CIn.Manager.Speed := 100;




           // Paletti Interni
           #PalettiInterni_Testa.Cin.Manager.Work := NOT #PalettiInterni_Testa.COut.Work;
           #PalettiInterni_Coda.Cin.Manager.Work := NOT #PalettiInterni_Coda.COut.Work;

           // Paletti Esterni
           #PalettiEsterni_Testa.Cin.Manager.Work := NOT #PalettiEsterni_Testa.COut.Work;
           #PalettiEsterni_Coda.Cin.Manager.Work := NOT #PalettiEsterni_Coda.COut.Work;


           // Trasporto in posizione di Trasporto
           #Ax_Testa.CIn.Manager.MoveToPos := #PalettiInterni_Testa.COut.Work AND #PalettiEsterni_Testa.COut.Work AND #PalettiInterni_Coda.COut.Work AND #PalettiEsterni_Coda.COut.Work AND NOT #AxTesta_InPosDeposito
           AND #Ax_Testa.S120.Sts.AxisEnabled AND #Ax_Coda.S120.Sts.AxisEnabled AND #TON_CheckAxis.Q;
           #Ax_Coda.CIn.Manager.MoveToPos := #PalettiInterni_Testa.COut.Work AND #PalettiEsterni_Testa.COut.Work AND #PalettiInterni_Coda.COut.Work AND #PalettiEsterni_Coda.COut.Work AND NOT #AxCoda_InPosDeposito
           AND #Ax_Testa.S120.Sts.AxisEnabled AND #Ax_Coda.S120.Sts.AxisEnabled AND #TON_CheckAxis.Q;

           #Ax_Coda.CIn.Manager.Pos := #Ax_Testa.CIn.Manager.Pos := #Par_Mach.PosDeposito;




       ELSIF #Ctrl.OP_Prelievo AND #Sts.OP_Prelievo_Cnd THEN
           #Ax_Testa.CIn.Manager.Speed := #Ax_Coda.CIn.Manager.Speed := 100;
           IF NOT #CIn.CycleModeShortPiece THEN

               // Paletti Interni
               #PalettiInterni_Testa.Cin.Manager.Work := NOT #PalettiInterni_Testa.COut.Work;
               #PalettiInterni_Coda.Cin.Manager.Work := NOT #PalettiInterni_Coda.COut.Work;

               #Ax_Coda.CIn.Manager.Pos := #Ax_Testa.CIn.Manager.Pos := #Par_Mach.PosPrelievo;

               #Ax_Testa.CIn.Manager.MoveToPos := NOT #AxTesta_InPosPrelievo AND #PalettiInterni_Testa.COut.Work AND #PalettiInterni_Coda.COut.Work
               AND #PalettiEsterni_Testa.COut.Rest AND #PalettiEsterni_Testa.COut.Rest AND #Ax_Testa.S120.Sts.AxisEnabled AND #Ax_Coda.S120.Sts.AxisEnabled;
               ;

               #Ax_Coda.CIn.Manager.MoveToPos := NOT #AxCoda_InPosPrelievo AND #PalettiInterni_Testa.COut.Work AND #PalettiInterni_Coda.COut.Work
               AND #PalettiEsterni_Testa.COut.Rest AND #PalettiEsterni_Testa.COut.Rest AND #Ax_Testa.S120.Sts.AxisEnabled AND #Ax_Coda.S120.Sts.AxisEnabled;
               ;

               // Paletti Esterni
               #PalettiEsterni_Testa.Cin.Manager.Work := #Sts.InPosPrelievo AND #PalettiInterni_Testa.COut.Work AND #PalettiInterni_Coda.COut.Work AND NOT #PalettiEsterni_Testa.COut.Work;
               #PalettiEsterni_Coda.Cin.Manager.Work := #Sts.InPosPrelievo AND #PalettiInterni_Coda.COut.Work AND #PalettiInterni_Testa.COut.Work AND NOT #PalettiEsterni_Coda.COut.Work;

           ELSE
               #Ax_Coda.CIn.Manager.Pos := #Ax_Testa.CIn.Manager.Pos := #Par_Mach.PosPrelievo;

               #Ax_Testa.CIn.Manager.MoveToPos := NOT #AxTesta_InPosPrelievo AND #PalettiInterni_Testa.COut.Rest AND #PalettiInterni_Coda.COut.Rest
               AND #PalettiEsterni_Testa.COut.Rest AND #PalettiEsterni_Testa.COut.Rest AND #Ax_Testa.S120.Sts.AxisEnabled AND #Ax_Coda.S120.Sts.AxisEnabled AND #TON_CheckAxis.Q;
               ;

               #Ax_Coda.CIn.Manager.MoveToPos := NOT #AxCoda_InPosPrelievo AND #PalettiInterni_Testa.COut.Rest AND #PalettiInterni_Coda.COut.Rest
               AND #PalettiEsterni_Testa.COut.Rest AND #PalettiEsterni_Testa.COut.Rest AND #Ax_Testa.S120.Sts.AxisEnabled AND #Ax_Coda.S120.Sts.AxisEnabled AND #TON_CheckAxis.Q;
               ;

           END_IF;
       END_IF;

   END_IF;



   IF #Ctrl.OP_Deposito AND #Sts.OP_Deposito_Cnd THEN
       #PalettiEsterni_Testa.Cin.Manager.Rest := NOT  #PalettiEsterni_Testa.COut.Rest;
       #PalettiEsterni_Coda.Cin.Manager.Rest := NOT #PalettiEsterni_Coda.COut.Rest;
       #PalettiInterni_Testa.Cin.Manager.Rest := NOT #PalettiInterni_Testa.COut.Rest;
       #PalettiInterni_Coda.Cin.Manager.Rest := NOT #PalettiInterni_Coda.COut.Rest;

   ELSIF NOT #Ctrl.OP_Deposito AND NOT #Ctrl.OP_Prelievo AND NOT #Ctrl.OP_Vai_A_Prelievo AND NOT #Ctrl.OP_Vai_A_Deposito THEN
       // Reset Cmd
       #Ax_Testa.CIn.Manager.Minus := FALSE;
       #Ax_Coda.CIn.Manager.Minus := FALSE;
       #PalettiEsterni_Testa.Cin.Manager.Rest := FALSE;
       #PalettiEsterni_Coda.Cin.Manager.Rest := FALSE;
       #PalettiInterni_Testa.Cin.Manager.Rest := FALSE;
       #PalettiInterni_Coda.Cin.Manager.Rest := FALSE;

       #Ax_Testa.CIn.Manager.Plus := FALSE;
       #Ax_Coda.CIn.Manager.Plus := FALSE;
       #Ax_Testa.CIn.Manager.MoveToPos := FALSE;
       #Ax_Coda.CIn.Manager.MoveToPos := FALSE;
       #PalettiEsterni_Testa.Cin.Manager.Work := FALSE;
       #PalettiEsterni_Coda.Cin.Manager.Work := FALSE;
       #PalettiInterni_Testa.Cin.Manager.Work := FALSE;
       #PalettiInterni_Coda.Cin.Manager.Work := FALSE;

   END_IF;
END_REGION

REGION Network 28: <+>
END_REGION

REGION Network 29: Warning manacanza condizioni esecuzione OperazionI
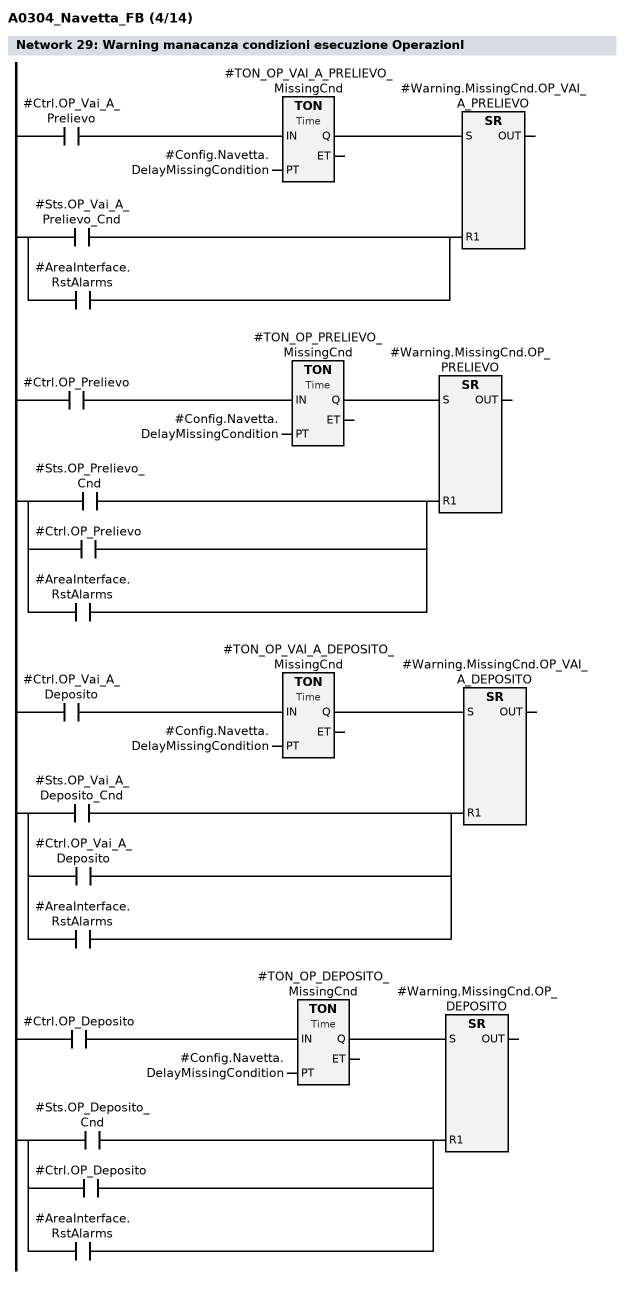
   RUNG wire#powerrail
      Contact( #Ctrl.OP_Vai_A_Prelievo )
      { S7_Templates := "time_type := Time" } #TON_OP_VAI_A_PRELIEVO_MissingCnd.TON(pt := #Config.Navetta.DelayMissingCondition, et =>)
      S_SR(operand := #Warning.MissingCnd.OP_VAI_A_PRELIEVO, r1 := wire#w1)
   END_RUNG
   RUNG wire#powerrail
      Contact( #Sts.OP_Vai_A_Prelievo_Cnd )
   END_RUNG wire#w1
   RUNG wire#powerrail
      Contact( #AreaInterface.RstAlarms )
   END_RUNG wire#w1
   RUNG wire#powerrail
      Contact( #Ctrl.OP_Prelievo )
      { S7_Templates := "time_type := Time" } #TON_OP_PRELIEVO_MissingCnd.TON(pt := #Config.Navetta.DelayMissingCondition, et =>)
      S_SR(operand := #Warning.MissingCnd.OP_PRELIEVO, r1 := wire#w2)
   END_RUNG
   RUNG wire#powerrail
      Contact( #Sts.OP_Prelievo_Cnd )
   END_RUNG wire#w2
   RUNG wire#powerrail
      Contact( #Ctrl.OP_Prelievo )
   END_RUNG wire#w2
   RUNG wire#powerrail
      Contact( #AreaInterface.RstAlarms )
   END_RUNG wire#w2
   RUNG wire#powerrail
      Contact( #Ctrl.OP_Vai_A_Deposito )
      { S7_Templates := "time_type := Time" } #TON_OP_VAI_A_DEPOSITO_MissingCnd.TON(pt := #Config.Navetta.DelayMissingCondition, et =>)
      S_SR(operand := #Warning.MissingCnd.OP_VAI_A_DEPOSITO, r1 := wire#w3)
   END_RUNG
   RUNG wire#powerrail
      Contact( #Sts.OP_Vai_A_Deposito_Cnd )
   END_RUNG wire#w3
   RUNG wire#powerrail
      Contact( #Ctrl.OP_Vai_A_Deposito )
   END_RUNG wire#w3
   RUNG wire#powerrail
      Contact( #AreaInterface.RstAlarms )
   END_RUNG wire#w3
   RUNG wire#powerrail
      Contact( #Ctrl.OP_Deposito )
      { S7_Templates := "time_type := Time" } #TON_OP_DEPOSITO_MissingCnd.TON(pt := #Config.Navetta.DelayMissingCondition, et =>)
      S_SR(operand := #Warning.MissingCnd.OP_DEPOSITO, r1 := wire#w4)
   END_RUNG
   RUNG wire#powerrail
      Contact( #Sts.OP_Deposito_Cnd )
   END_RUNG wire#w4
   RUNG wire#powerrail
      Contact( #Ctrl.OP_Deposito )
   END_RUNG wire#w4
   RUNG wire#powerrail
      Contact( #AreaInterface.RstAlarms )
   END_RUNG wire#w4
   // the same network as SCL:
   #TON_OP_VAI_A_PRELIEVO_MissingCnd.TON(IN := #Ctrl.OP_Vai_A_Prelievo,
                           PT := #Config.Navetta.DelayMissingCondition);
   IF #TON_OP_VAI_A_PRELIEVO_MissingCnd.Q THEN
       #Warning.MissingCnd.OP_VAI_A_PRELIEVO := TRUE;   // SR flip-flop
   END_IF;
   IF #Sts.OP_Vai_A_Prelievo_Cnd OR #AreaInterface.RstAlarms THEN
       #Warning.MissingCnd.OP_VAI_A_PRELIEVO := FALSE;
   END_IF;
   #TON_OP_PRELIEVO_MissingCnd.TON(IN := #Ctrl.OP_Prelievo, PT := #Config.Navetta.DelayMissingCondition);
   IF #TON_OP_PRELIEVO_MissingCnd.Q THEN
       #Warning.MissingCnd.OP_PRELIEVO := TRUE;   // SR flip-flop
   END_IF;
   IF #Sts.OP_Prelievo_Cnd OR #Ctrl.OP_Prelievo OR #AreaInterface.RstAlarms THEN
       #Warning.MissingCnd.OP_PRELIEVO := FALSE;
   END_IF;
   #TON_OP_VAI_A_DEPOSITO_MissingCnd.TON(IN := #Ctrl.OP_Vai_A_Deposito,
                           PT := #Config.Navetta.DelayMissingCondition);
   IF #TON_OP_VAI_A_DEPOSITO_MissingCnd.Q THEN
       #Warning.MissingCnd.OP_VAI_A_DEPOSITO := TRUE;   // SR flip-flop
   END_IF;
   IF #Sts.OP_Vai_A_Deposito_Cnd OR #Ctrl.OP_Vai_A_Deposito OR #AreaInterface.RstAlarms THEN
       #Warning.MissingCnd.OP_VAI_A_DEPOSITO := FALSE;
   END_IF;
   #TON_OP_DEPOSITO_MissingCnd.TON(IN := #Ctrl.OP_Deposito, PT := #Config.Navetta.DelayMissingCondition);
   IF #TON_OP_DEPOSITO_MissingCnd.Q THEN
       #Warning.MissingCnd.OP_DEPOSITO := TRUE;   // SR flip-flop
   END_IF;
   IF #Sts.OP_Deposito_Cnd OR #Ctrl.OP_Deposito OR #AreaInterface.RstAlarms THEN
       #Warning.MissingCnd.OP_DEPOSITO := FALSE;
   END_IF;
END_REGION

REGION Network 30 (SCL): Shuttle Out of Workspace
   IF #Ax_Coda.COut.ActualPosition > #"Ax_Fuori Ingombro" AND #Ax_Testa.COut.ActualPosition > #"Ax_Fuori Ingombro" THEN
       #Sts.OutOfWorkSpace := TRUE;
   ELSE
       #Sts.OutOfWorkSpace := FALSE;
   END_IF;
END_REGION

REGION Network 31: Check Shuttle Movement
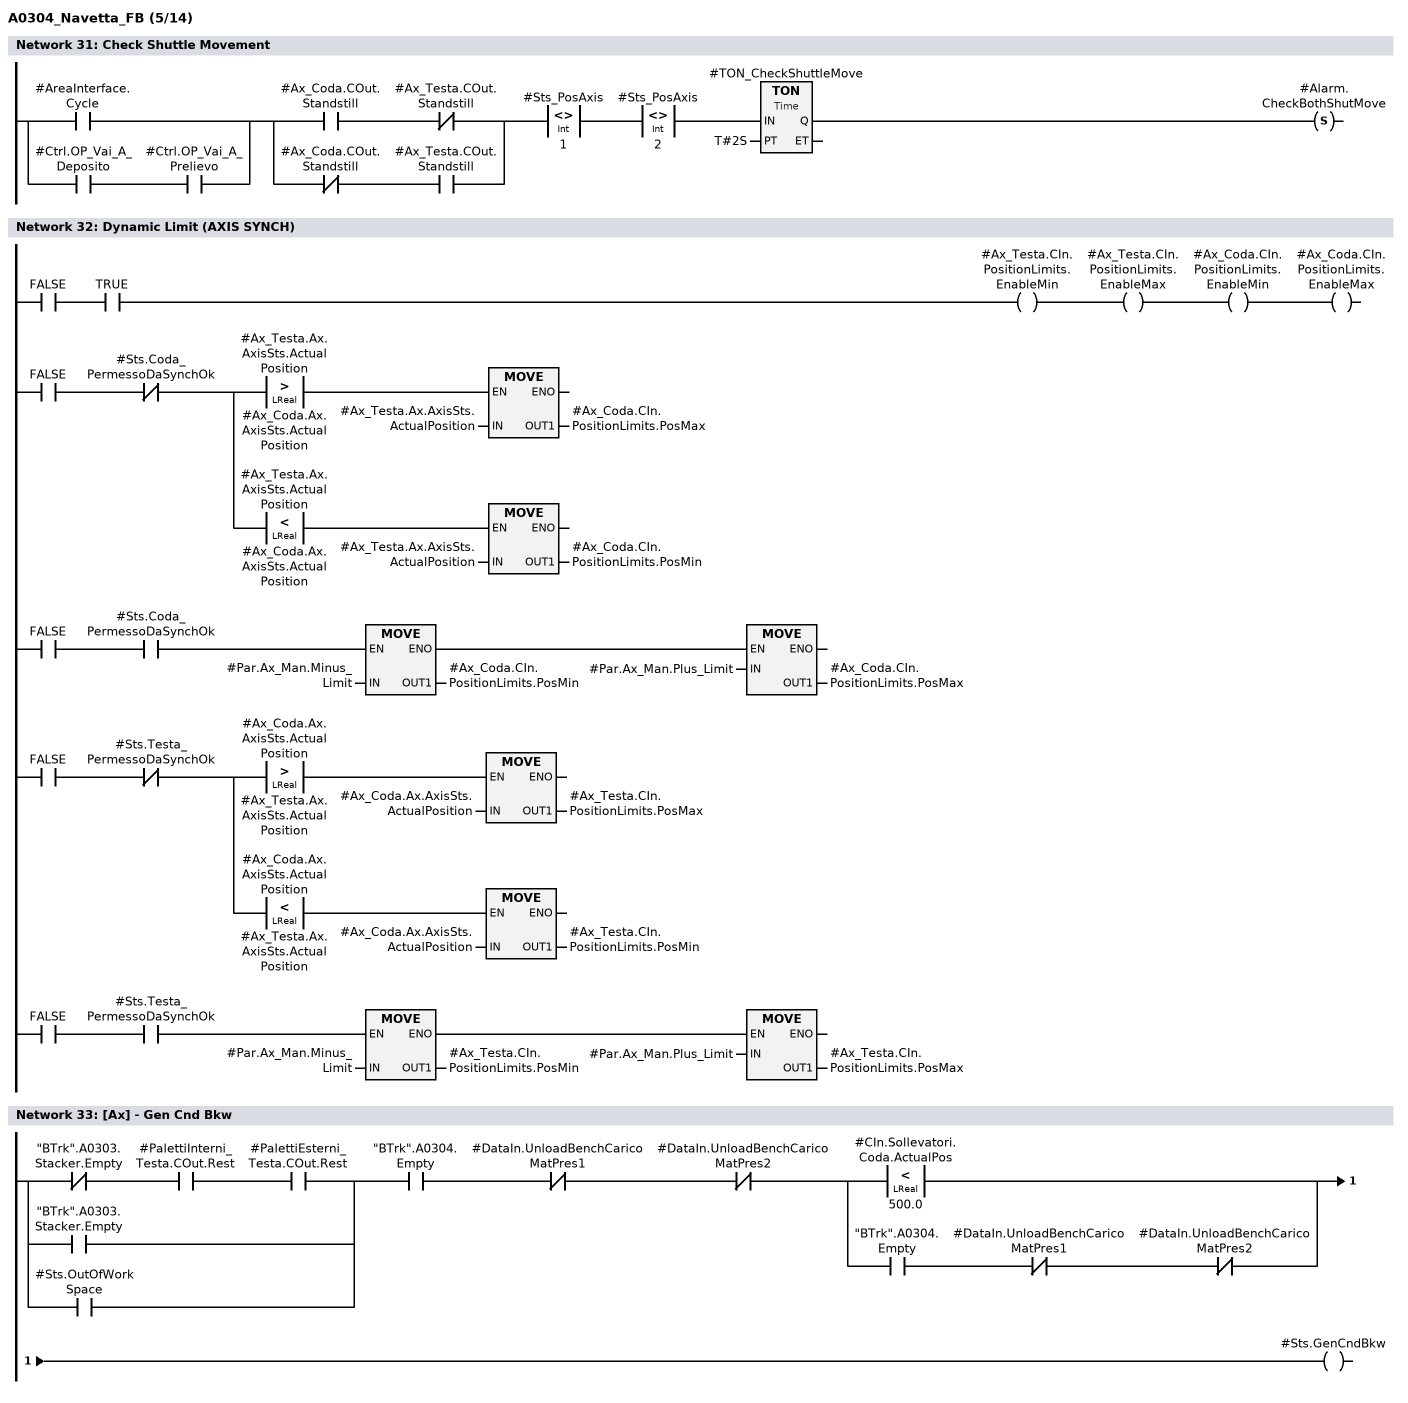
   RUNG wire#powerrail
      Contact( #AreaInterface.Cycle )
      wire#w1
      Contact( #Ax_Coda.COut.Standstill )
      I_Contact( #Ax_Testa.COut.Standstill )
      wire#w2
      { S7_Templates := "SrcType := Int" } NE_Contact(in1 := #Sts_PosAxis, in2 := 1)
      { S7_Templates := "SrcType := Int" } NE_Contact(in1 := #Sts_PosAxis, in2 := 2)
      { S7_Templates := "time_type := Time" } #TON_CheckShuttleMove.TON(pt := T#2S, et =>)
      S_Coil( #Alarm.CheckBothShutMove )
   END_RUNG
   RUNG wire#powerrail
      Contact( #Ctrl.OP_Vai_A_Deposito )
      Contact( #Ctrl.OP_Vai_A_Prelievo )
   END_RUNG wire#w1
   RUNG wire#w1
      I_Contact( #Ax_Coda.COut.Standstill )
      Contact( #Ax_Testa.COut.Standstill )
   END_RUNG wire#w2
   // the same network as SCL:
   #TON_CheckShuttleMove.TON(IN := (#AreaInterface.Cycle OR (#Ctrl.OP_Vai_A_Deposito AND #Ctrl.OP_Vai_A_Prelievo)) AND ((#Ax_Coda.COut.Standstill AND NOT #Ax_Testa.COut.Standstill) OR (NOT #Ax_Coda.COut.Standstill AND #Ax_Testa.COut.Standstill)) AND (#Sts_PosAxis <> 1) AND (#Sts_PosAxis <> 2),
                           PT := T#2S);
   IF #TON_CheckShuttleMove.Q THEN #Alarm.CheckBothShutMove := TRUE; END_IF;
END_REGION

REGION Network 32: Dynamic Limit (AXIS SYNCH)
   RUNG wire#powerrail
      Contact( FALSE )
      Contact( TRUE )
      Coil( #Ax_Testa.CIn.PositionLimits.EnableMin )
      Coil( #Ax_Testa.CIn.PositionLimits.EnableMax )
      Coil( #Ax_Coda.CIn.PositionLimits.EnableMin )
      Coil( #Ax_Coda.CIn.PositionLimits.EnableMax )
   END_RUNG
   RUNG wire#powerrail
      Contact( FALSE )
      I_Contact( #Sts.Coda_PermessoDaSynchOk )
      wire#w1
      { S7_Templates := "SrcType := LReal" } GT_Contact(in1 := #Ax_Testa.Ax.AxisSts.ActualPosition, in2 := #Ax_Coda.Ax.AxisSts.ActualPosition)
      Move(in := #Ax_Testa.Ax.AxisSts.ActualPosition, out1 => #Ax_Coda.CIn.PositionLimits.PosMax)
   END_RUNG
   RUNG wire#w1
      { S7_Templates := "SrcType := LReal" } LT_Contact(in1 := #Ax_Testa.Ax.AxisSts.ActualPosition, in2 := #Ax_Coda.Ax.AxisSts.ActualPosition)
      Move(in := #Ax_Testa.Ax.AxisSts.ActualPosition, out1 => #Ax_Coda.CIn.PositionLimits.PosMin)
   END_RUNG
   RUNG wire#powerrail
      Contact( FALSE )
      Contact( #Sts.Coda_PermessoDaSynchOk )
      Move(in := #Par.Ax_Man.Minus_Limit, out1 => #Ax_Coda.CIn.PositionLimits.PosMin)
      Move(in := #Par.Ax_Man.Plus_Limit, out1 => #Ax_Coda.CIn.PositionLimits.PosMax)
   END_RUNG
   RUNG wire#powerrail
      Contact( FALSE )
      I_Contact( #Sts.Testa_PermessoDaSynchOk )
      wire#w2
      { S7_Templates := "SrcType := LReal" } GT_Contact(in1 := #Ax_Coda.Ax.AxisSts.ActualPosition, in2 := #Ax_Testa.Ax.AxisSts.ActualPosition)
      Move(in := #Ax_Coda.Ax.AxisSts.ActualPosition, out1 => #Ax_Testa.CIn.PositionLimits.PosMax)
   END_RUNG
   RUNG wire#w2
      { S7_Templates := "SrcType := LReal" } LT_Contact(in1 := #Ax_Coda.Ax.AxisSts.ActualPosition, in2 := #Ax_Testa.Ax.AxisSts.ActualPosition)
      Move(in := #Ax_Coda.Ax.AxisSts.ActualPosition, out1 => #Ax_Testa.CIn.PositionLimits.PosMin)
   END_RUNG
   RUNG wire#powerrail
      Contact( FALSE )
      Contact( #Sts.Testa_PermessoDaSynchOk )
      Move(in := #Par.Ax_Man.Minus_Limit, out1 => #Ax_Testa.CIn.PositionLimits.PosMin)
      Move(in := #Par.Ax_Man.Plus_Limit, out1 => #Ax_Testa.CIn.PositionLimits.PosMax)
   END_RUNG
   // the same network as SCL:
   #Ax_Testa.CIn.PositionLimits.EnableMin := FALSE AND TRUE;
   #Ax_Testa.CIn.PositionLimits.EnableMax := #Ax_Testa.CIn.PositionLimits.EnableMin;
   #Ax_Coda.CIn.PositionLimits.EnableMin := #Ax_Testa.CIn.PositionLimits.EnableMin;
   #Ax_Coda.CIn.PositionLimits.EnableMax := #Ax_Testa.CIn.PositionLimits.EnableMin;
   #_w1 := FALSE AND NOT #Sts.Coda_PermessoDaSynchOk;
   IF #_w1 AND (#Ax_Testa.Ax.AxisSts.ActualPosition > #Ax_Coda.Ax.AxisSts.ActualPosition) THEN
       #Ax_Coda.CIn.PositionLimits.PosMax := #Ax_Testa.Ax.AxisSts.ActualPosition;
   END_IF;
   IF #_w1 AND (#Ax_Testa.Ax.AxisSts.ActualPosition < #Ax_Coda.Ax.AxisSts.ActualPosition) THEN
       #Ax_Coda.CIn.PositionLimits.PosMin := #Ax_Testa.Ax.AxisSts.ActualPosition;
   END_IF;
   IF FALSE AND #Sts.Coda_PermessoDaSynchOk THEN
       #Ax_Coda.CIn.PositionLimits.PosMin := #Par.Ax_Man.Minus_Limit;
       #Ax_Coda.CIn.PositionLimits.PosMax := #Par.Ax_Man.Plus_Limit;
   END_IF;
   #_w2 := FALSE AND NOT #Sts.Testa_PermessoDaSynchOk;
   IF #_w2 AND (#Ax_Coda.Ax.AxisSts.ActualPosition > #Ax_Testa.Ax.AxisSts.ActualPosition) THEN
       #Ax_Testa.CIn.PositionLimits.PosMax := #Ax_Coda.Ax.AxisSts.ActualPosition;
   END_IF;
   IF #_w2 AND (#Ax_Coda.Ax.AxisSts.ActualPosition < #Ax_Testa.Ax.AxisSts.ActualPosition) THEN
       #Ax_Testa.CIn.PositionLimits.PosMin := #Ax_Coda.Ax.AxisSts.ActualPosition;
   END_IF;
   IF FALSE AND #Sts.Testa_PermessoDaSynchOk THEN
       #Ax_Testa.CIn.PositionLimits.PosMin := #Par.Ax_Man.Minus_Limit;
       #Ax_Testa.CIn.PositionLimits.PosMax := #Par.Ax_Man.Plus_Limit;
   END_IF;
END_REGION

REGION Network 33: [Ax] - Gen Cnd Bkw
   RUNG wire#powerrail
      I_Contact( "BTrk".A0303.Stacker.Empty )
      Contact( #PalettiInterni_Testa.COut.Rest )
      Contact( #PalettiEsterni_Testa.COut.Rest )
      wire#w1
      Contact( "BTrk".A0304.Empty )
      I_Contact( #DataIn.UnloadBenchCaricoMatPres1 )
      I_Contact( #DataIn.UnloadBenchCaricoMatPres2 )
      wire#w2
      { S7_Templates := "SrcType := LReal" } LT_Contact(in1 := #CIn.Sollevatori.Coda.ActualPos, in2 := 500.0)
      wire#w3
      Coil( #Sts.GenCndBkw )
   END_RUNG
   RUNG wire#powerrail
      Contact( "BTrk".A0303.Stacker.Empty )
   END_RUNG wire#w1
   RUNG wire#powerrail
      Contact( #Sts.OutOfWorkSpace )
   END_RUNG wire#w1
   RUNG wire#w2
      Contact( "BTrk".A0304.Empty )
      I_Contact( #DataIn.UnloadBenchCaricoMatPres1 )
      I_Contact( #DataIn.UnloadBenchCaricoMatPres2 )
   END_RUNG wire#w3
   // the same network as SCL:
   #Sts.GenCndBkw := ((NOT "BTrk".A0303.Stacker.Empty AND #PalettiInterni_Testa.COut.Rest AND #PalettiEsterni_Testa.COut.Rest) OR "BTrk".A0303.Stacker.Empty OR #Sts.OutOfWorkSpace) AND "BTrk".A0304.Empty AND NOT #DataIn.UnloadBenchCaricoMatPres1 AND NOT #DataIn.UnloadBenchCaricoMatPres2 AND ((#CIn.Sollevatori.Coda.ActualPos < 500.0) OR ("BTrk".A0304.Empty AND NOT #DataIn.UnloadBenchCaricoMatPres1 AND NOT #DataIn.UnloadBenchCaricoMatPres2));
END_REGION

REGION Network 34: [Ax] - Gen Cnd Fwd
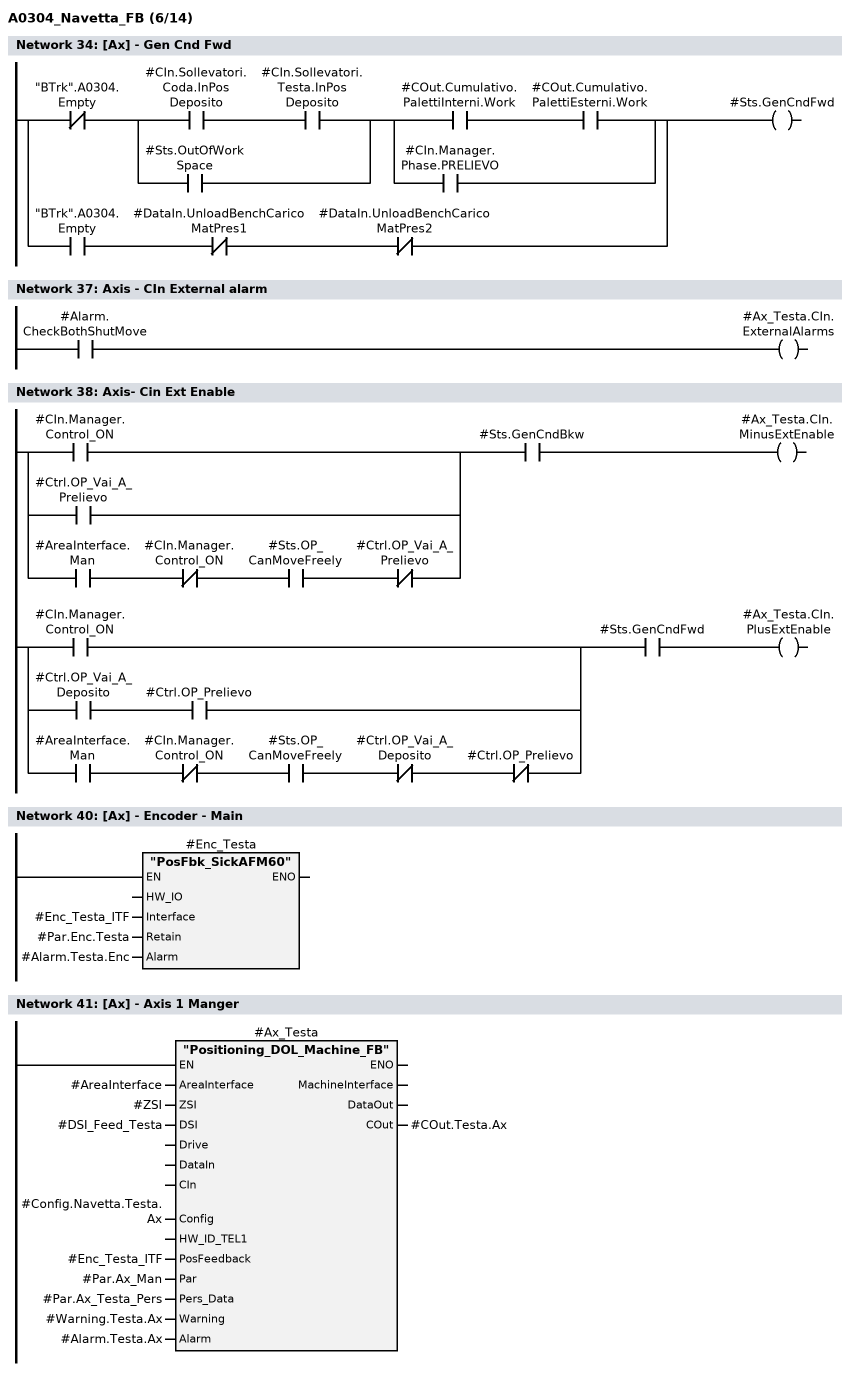
   RUNG wire#powerrail
      I_Contact( "BTrk".A0304.Empty )
      wire#w1
      Contact( #CIn.Sollevatori.Coda.InPosDeposito )
      Contact( #CIn.Sollevatori.Testa.InPosDeposito )
      wire#w2
      Contact( #COut.Cumulativo.PalettiInterni.Work )
      Contact( #COut.Cumulativo.PalettiEsterni.Work )
      wire#w3
      Coil( #Sts.GenCndFwd )
   END_RUNG
   RUNG wire#w1
      Contact( #Sts.OutOfWorkSpace )
   END_RUNG wire#w2
   RUNG wire#w2
      Contact( #CIn.Manager.Phase.PRELIEVO )
   END_RUNG wire#w3
   RUNG wire#powerrail
      Contact( "BTrk".A0304.Empty )
      I_Contact( #DataIn.UnloadBenchCaricoMatPres1 )
      I_Contact( #DataIn.UnloadBenchCaricoMatPres2 )
   END_RUNG wire#w3
   // the same network as SCL:
   #Sts.GenCndFwd := (NOT "BTrk".A0304.Empty AND ((#CIn.Sollevatori.Coda.InPosDeposito AND #CIn.Sollevatori.Testa.InPosDeposito) OR #Sts.OutOfWorkSpace) AND ((#COut.Cumulativo.PalettiInterni.Work AND #COut.Cumulativo.PalettiEsterni.Work) OR #CIn.Manager.Phase.PRELIEVO)) OR ("BTrk".A0304.Empty AND NOT #DataIn.UnloadBenchCaricoMatPres1 AND NOT #DataIn.UnloadBenchCaricoMatPres2);
END_REGION

REGION Network 35: <<<<<<<<<<<<<<<<<<<<<<<<<<<<<<<<<< LATO TESTA >>>>>>>>>>>>>>>>>>>>>>>>>>>>>>>>>>>>>>>
END_REGION

REGION Network 36: <<< ASSE >>>
END_REGION

REGION Network 37: Axis - CIn External alarm
   RUNG wire#powerrail
      Contact( #Alarm.CheckBothShutMove )
      Coil( #Ax_Testa.CIn.ExternalAlarms )
   END_RUNG
   // the same network as SCL:
   #Ax_Testa.CIn.ExternalAlarms := #Alarm.CheckBothShutMove;
END_REGION

REGION Network 38: Axis- Cin Ext Enable
   RUNG wire#powerrail
      Contact( #CIn.Manager.Control_ON )
      wire#w1
      Contact( #Sts.GenCndBkw )
      Coil( #Ax_Testa.CIn.MinusExtEnable )
   END_RUNG
   RUNG wire#powerrail
      Contact( #Ctrl.OP_Vai_A_Prelievo )
   END_RUNG wire#w1
   RUNG wire#powerrail
      Contact( #AreaInterface.Man )
      I_Contact( #CIn.Manager.Control_ON )
      Contact( #Sts.OP_CanMoveFreely )
      I_Contact( #Ctrl.OP_Vai_A_Prelievo )
   END_RUNG wire#w1
   RUNG wire#powerrail
      Contact( #CIn.Manager.Control_ON )
      wire#w2
      Contact( #Sts.GenCndFwd )
      Coil( #Ax_Testa.CIn.PlusExtEnable )
   END_RUNG
   RUNG wire#powerrail
      Contact( #Ctrl.OP_Vai_A_Deposito )
      Contact( #Ctrl.OP_Prelievo )
   END_RUNG wire#w2
   RUNG wire#powerrail
      Contact( #AreaInterface.Man )
      I_Contact( #CIn.Manager.Control_ON )
      Contact( #Sts.OP_CanMoveFreely )
      I_Contact( #Ctrl.OP_Vai_A_Deposito )
      I_Contact( #Ctrl.OP_Prelievo )
   END_RUNG wire#w2
   // the same network as SCL:
   #Ax_Testa.CIn.MinusExtEnable := (#CIn.Manager.Control_ON OR #Ctrl.OP_Vai_A_Prelievo OR (#AreaInterface.Man AND NOT #CIn.Manager.Control_ON AND #Sts.OP_CanMoveFreely AND NOT #Ctrl.OP_Vai_A_Prelievo)) AND #Sts.GenCndBkw;
   #Ax_Testa.CIn.PlusExtEnable := (#CIn.Manager.Control_ON OR (#Ctrl.OP_Vai_A_Deposito AND #Ctrl.OP_Prelievo) OR (#AreaInterface.Man AND NOT #CIn.Manager.Control_ON AND #Sts.OP_CanMoveFreely AND NOT #Ctrl.OP_Vai_A_Deposito AND NOT #Ctrl.OP_Prelievo)) AND #Sts.GenCndFwd;
END_REGION

REGION Network 39 (SCL): HMI preset position
   #Ax_Testa.HMI.B_Preset := #HMI.Testa.PbPreset;

   #Ax_Testa.HMI.PresetPosition := #HMI.Testa.PresetValue;
END_REGION

REGION Network 40: [Ax] - Encoder - Main
   RUNG wire#powerrail
      #Enc_Testa(HW_IO :=, Interface := #Enc_Testa_ITF, Retain := #Par.Enc.Testa, Alarm := #Alarm.Testa.Enc)
   END_RUNG
   // the same network as SCL:
   #Enc_Testa(Interface := #Enc_Testa_ITF, Retain := #Par.Enc.Testa, Alarm := #Alarm.Testa.Enc);   // "PosFbk_SickAFM60"
END_REGION

REGION Network 41: [Ax] - Axis 1 Manger
   RUNG wire#powerrail
      #Ax_Testa(AreaInterface := #AreaInterface, ZSI := #ZSI, DSI := #DSI_Feed_Testa, Drive :=, DataIn :=, CIn :=, Config := #Config.Navetta.Testa.Ax, HW_ID_TEL1 :=, PosFeedback := #Enc_Testa_ITF, Par := #Par.Ax_Man, Pers_Data := #Par.Ax_Testa_Pers, Warning := #Warning.Testa.Ax, Alarm := #Alarm.Testa.Ax, MachineInterface =>, DataOut =>, COut => #COut.Testa.Ax)
   END_RUNG
   // the same network as SCL:
   #Ax_Testa(AreaInterface := #AreaInterface,   // "Positioning_DOL_Machine_FB"
             ZSI := #ZSI,
             DSI := #DSI_Feed_Testa,
             Config := #Config.Navetta.Testa.Ax,
             PosFeedback := #Enc_Testa_ITF,
             Par := #Par.Ax_Man,
             Pers_Data := #Par.Ax_Testa_Pers,
             Warning := #Warning.Testa.Ax,
             Alarm := #Alarm.Testa.Ax,
             COut => #COut.Testa.Ax);
END_REGION

REGION Network 43: <<< PALETTI INTRENI >>>
END_REGION

REGION Network 44: Paletti Interni - CIn External alarm
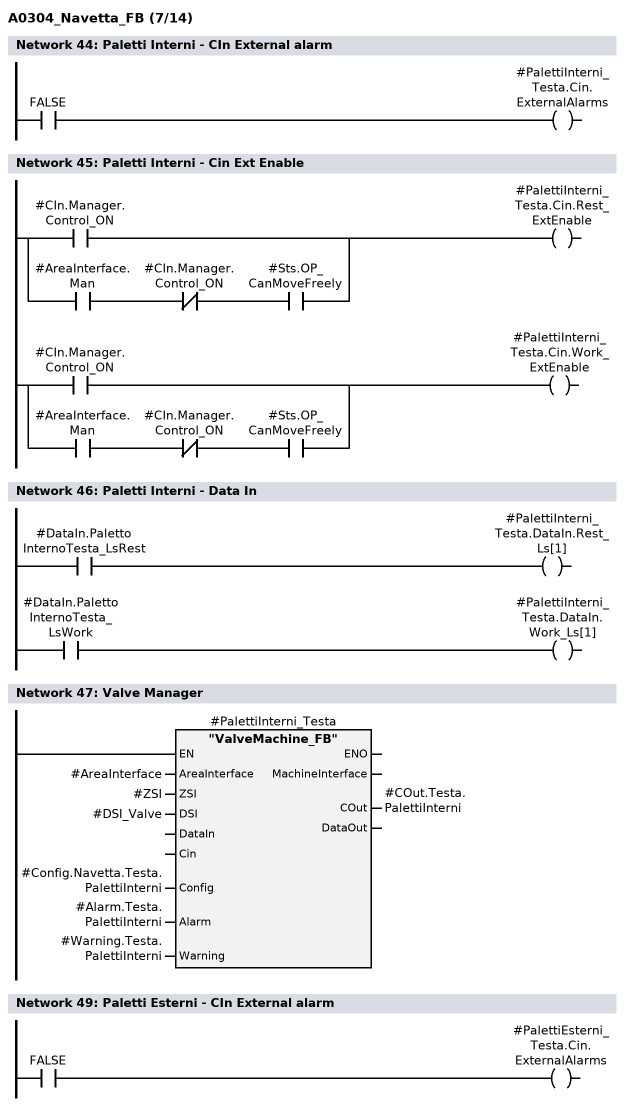
   RUNG wire#powerrail
      Contact( FALSE )
      Coil( #PalettiInterni_Testa.Cin.ExternalAlarms )
   END_RUNG
   // the same network as SCL:
   #PalettiInterni_Testa.Cin.ExternalAlarms := FALSE;
END_REGION

REGION Network 45: Paletti Interni - Cin Ext Enable
   RUNG wire#powerrail
      Contact( #CIn.Manager.Control_ON )
      wire#w1
      Coil( #PalettiInterni_Testa.Cin.Rest_ExtEnable )
   END_RUNG
   RUNG wire#powerrail
      Contact( #AreaInterface.Man )
      I_Contact( #CIn.Manager.Control_ON )
      Contact( #Sts.OP_CanMoveFreely )
   END_RUNG wire#w1
   RUNG wire#powerrail
      Contact( #CIn.Manager.Control_ON )
      wire#w2
      Coil( #PalettiInterni_Testa.Cin.Work_ExtEnable )
   END_RUNG
   RUNG wire#powerrail
      Contact( #AreaInterface.Man )
      I_Contact( #CIn.Manager.Control_ON )
      Contact( #Sts.OP_CanMoveFreely )
   END_RUNG wire#w2
   // the same network as SCL:
   #PalettiInterni_Testa.Cin.Rest_ExtEnable := #CIn.Manager.Control_ON OR (#AreaInterface.Man AND NOT #CIn.Manager.Control_ON AND #Sts.OP_CanMoveFreely);
   #PalettiInterni_Testa.Cin.Work_ExtEnable := #CIn.Manager.Control_ON OR (#AreaInterface.Man AND NOT #CIn.Manager.Control_ON AND #Sts.OP_CanMoveFreely);
END_REGION

REGION Network 46: Paletti Interni - Data In
   RUNG wire#powerrail
      Contact( #DataIn.PalettoInternoTesta_LsRest )
      Coil( #PalettiInterni_Testa.DataIn.Rest_Ls[1] )
   END_RUNG
   RUNG wire#powerrail
      Contact( #DataIn.PalettoInternoTesta_LsWork )
      Coil( #PalettiInterni_Testa.DataIn.Work_Ls[1] )
   END_RUNG
   // the same network as SCL:
   #PalettiInterni_Testa.DataIn.Rest_Ls[1] := #DataIn.PalettoInternoTesta_LsRest;
   #PalettiInterni_Testa.DataIn.Work_Ls[1] := #DataIn.PalettoInternoTesta_LsWork;
END_REGION

REGION Network 47: Valve Manager
   RUNG wire#powerrail
      #PalettiInterni_Testa(AreaInterface := #AreaInterface, ZSI := #ZSI, DSI := #DSI_Valve, DataIn :=, Cin :=, Config := #Config.Navetta.Testa.PalettiInterni, Alarm := #Alarm.Testa.PalettiInterni, Warning := #Warning.Testa.PalettiInterni, MachineInterface =>, COut => #COut.Testa.PalettiInterni, DataOut =>)
   END_RUNG
   // the same network as SCL:
   #PalettiInterni_Testa(AreaInterface := #AreaInterface,   // "ValveMachine_FB"
                         ZSI := #ZSI,
                         DSI := #DSI_Valve,
                         Config := #Config.Navetta.Testa.PalettiInterni,
                         Alarm := #Alarm.Testa.PalettiInterni,
                         Warning := #Warning.Testa.PalettiInterni,
                         COut => #COut.Testa.PalettiInterni);
END_REGION

REGION Network 48: <<< PALETTI ESTERNI>>>
END_REGION

REGION Network 49: Paletti Esterni - CIn External alarm
   RUNG wire#powerrail
      Contact( FALSE )
      Coil( #PalettiEsterni_Testa.Cin.ExternalAlarms )
   END_RUNG
   // the same network as SCL:
   #PalettiEsterni_Testa.Cin.ExternalAlarms := FALSE;
END_REGION

REGION Network 50: Paletti Esterni - Cin Ext Enable
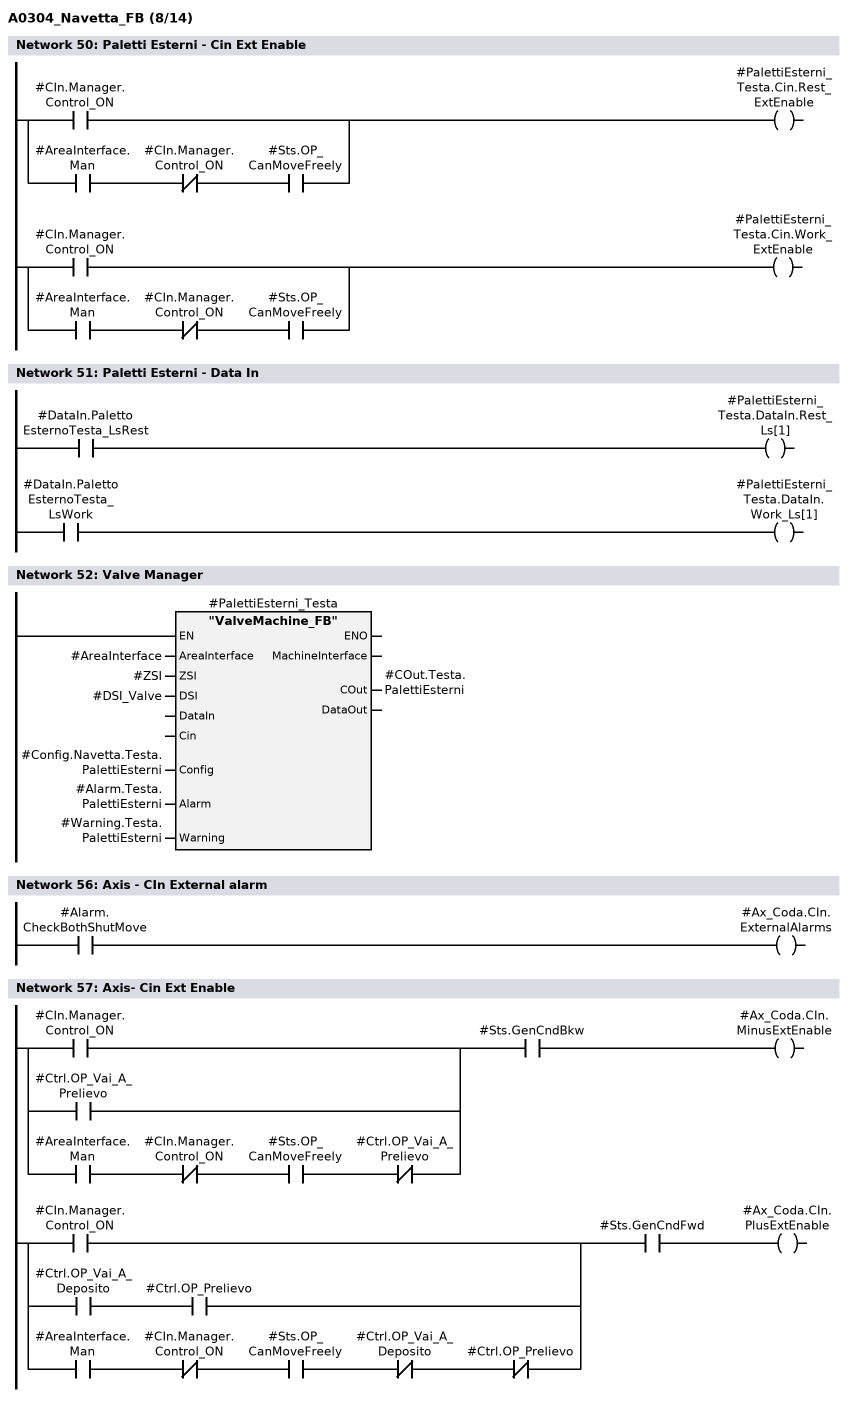
   RUNG wire#powerrail
      Contact( #CIn.Manager.Control_ON )
      wire#w1
      Coil( #PalettiEsterni_Testa.Cin.Rest_ExtEnable )
   END_RUNG
   RUNG wire#powerrail
      Contact( #AreaInterface.Man )
      I_Contact( #CIn.Manager.Control_ON )
      Contact( #Sts.OP_CanMoveFreely )
   END_RUNG wire#w1
   RUNG wire#powerrail
      Contact( #CIn.Manager.Control_ON )
      wire#w2
      Coil( #PalettiEsterni_Testa.Cin.Work_ExtEnable )
   END_RUNG
   RUNG wire#powerrail
      Contact( #AreaInterface.Man )
      I_Contact( #CIn.Manager.Control_ON )
      Contact( #Sts.OP_CanMoveFreely )
   END_RUNG wire#w2
   // the same network as SCL:
   #PalettiEsterni_Testa.Cin.Rest_ExtEnable := #CIn.Manager.Control_ON OR (#AreaInterface.Man AND NOT #CIn.Manager.Control_ON AND #Sts.OP_CanMoveFreely);
   #PalettiEsterni_Testa.Cin.Work_ExtEnable := #CIn.Manager.Control_ON OR (#AreaInterface.Man AND NOT #CIn.Manager.Control_ON AND #Sts.OP_CanMoveFreely);
END_REGION

REGION Network 51: Paletti Esterni - Data In
   RUNG wire#powerrail
      Contact( #DataIn.PalettoEsternoTesta_LsRest )
      Coil( #PalettiEsterni_Testa.DataIn.Rest_Ls[1] )
   END_RUNG
   RUNG wire#powerrail
      Contact( #DataIn.PalettoEsternoTesta_LsWork )
      Coil( #PalettiEsterni_Testa.DataIn.Work_Ls[1] )
   END_RUNG
   // the same network as SCL:
   #PalettiEsterni_Testa.DataIn.Rest_Ls[1] := #DataIn.PalettoEsternoTesta_LsRest;
   #PalettiEsterni_Testa.DataIn.Work_Ls[1] := #DataIn.PalettoEsternoTesta_LsWork;
END_REGION

REGION Network 52: Valve Manager
   RUNG wire#powerrail
      #PalettiEsterni_Testa(AreaInterface := #AreaInterface, ZSI := #ZSI, DSI := #DSI_Valve, DataIn :=, Cin :=, Config := #Config.Navetta.Testa.PalettiEsterni, Alarm := #Alarm.Testa.PalettiEsterni, Warning := #Warning.Testa.PalettiEsterni, MachineInterface =>, COut => #COut.Testa.PalettiEsterni, DataOut =>)
   END_RUNG
   // the same network as SCL:
   #PalettiEsterni_Testa(AreaInterface := #AreaInterface,   // "ValveMachine_FB"
                         ZSI := #ZSI,
                         DSI := #DSI_Valve,
                         Config := #Config.Navetta.Testa.PalettiEsterni,
                         Alarm := #Alarm.Testa.PalettiEsterni,
                         Warning := #Warning.Testa.PalettiEsterni,
                         COut => #COut.Testa.PalettiEsterni);
END_REGION

REGION Network 54: <<<<<<<<<<<<<<<<<<<<<<<<<<<<<<<<<< LATO CODA >>>>>>>>>>>>>>>>>>>>>>>>>>>>>>>>>>>>>>>
END_REGION

REGION Network 55: <<< ASSE >>>
END_REGION

REGION Network 56: Axis - CIn External alarm
   RUNG wire#powerrail
      Contact( #Alarm.CheckBothShutMove )
      Coil( #Ax_Coda.CIn.ExternalAlarms )
   END_RUNG
   // the same network as SCL:
   #Ax_Coda.CIn.ExternalAlarms := #Alarm.CheckBothShutMove;
END_REGION

REGION Network 57: Axis- Cin Ext Enable
   RUNG wire#powerrail
      Contact( #CIn.Manager.Control_ON )
      wire#w1
      Contact( #Sts.GenCndBkw )
      Coil( #Ax_Coda.CIn.MinusExtEnable )
   END_RUNG
   RUNG wire#powerrail
      Contact( #Ctrl.OP_Vai_A_Prelievo )
   END_RUNG wire#w1
   RUNG wire#powerrail
      Contact( #AreaInterface.Man )
      I_Contact( #CIn.Manager.Control_ON )
      Contact( #Sts.OP_CanMoveFreely )
      I_Contact( #Ctrl.OP_Vai_A_Prelievo )
   END_RUNG wire#w1
   RUNG wire#powerrail
      Contact( #CIn.Manager.Control_ON )
      wire#w2
      Contact( #Sts.GenCndFwd )
      Coil( #Ax_Coda.CIn.PlusExtEnable )
   END_RUNG
   RUNG wire#powerrail
      Contact( #Ctrl.OP_Vai_A_Deposito )
      Contact( #Ctrl.OP_Prelievo )
   END_RUNG wire#w2
   RUNG wire#powerrail
      Contact( #AreaInterface.Man )
      I_Contact( #CIn.Manager.Control_ON )
      Contact( #Sts.OP_CanMoveFreely )
      I_Contact( #Ctrl.OP_Vai_A_Deposito )
      I_Contact( #Ctrl.OP_Prelievo )
   END_RUNG wire#w2
   // the same network as SCL:
   #Ax_Coda.CIn.MinusExtEnable := (#CIn.Manager.Control_ON OR #Ctrl.OP_Vai_A_Prelievo OR (#AreaInterface.Man AND NOT #CIn.Manager.Control_ON AND #Sts.OP_CanMoveFreely AND NOT #Ctrl.OP_Vai_A_Prelievo)) AND #Sts.GenCndBkw;
   #Ax_Coda.CIn.PlusExtEnable := (#CIn.Manager.Control_ON OR (#Ctrl.OP_Vai_A_Deposito AND #Ctrl.OP_Prelievo) OR (#AreaInterface.Man AND NOT #CIn.Manager.Control_ON AND #Sts.OP_CanMoveFreely AND NOT #Ctrl.OP_Vai_A_Deposito AND NOT #Ctrl.OP_Prelievo)) AND #Sts.GenCndFwd;
END_REGION

REGION Network 58 (SCL): HMI preset position
   #Ax_Coda.HMI.B_Preset := #HMI.Coda.PbPreset;

   #Ax_Coda.HMI.PresetPosition := #HMI.Coda.PresetValue;
END_REGION

REGION Network 59: [Ax] - Encoder - Main
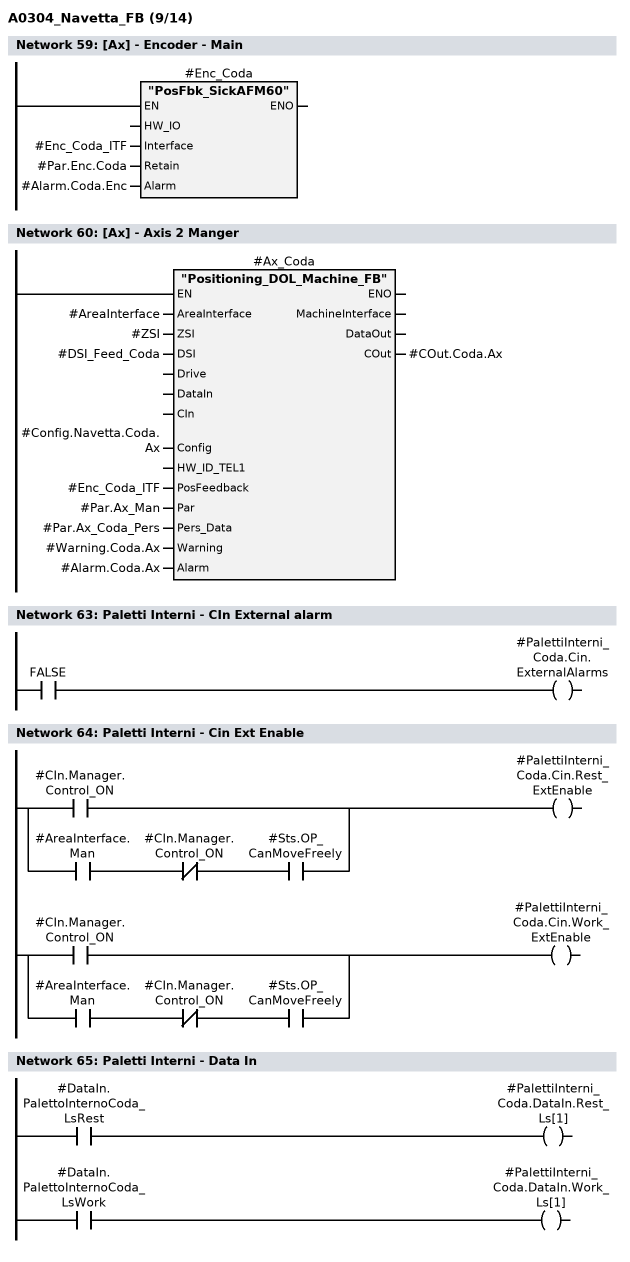
   RUNG wire#powerrail
      #Enc_Coda(HW_IO :=, Interface := #Enc_Coda_ITF, Retain := #Par.Enc.Coda, Alarm := #Alarm.Coda.Enc)
   END_RUNG
   // the same network as SCL:
   #Enc_Coda(Interface := #Enc_Coda_ITF, Retain := #Par.Enc.Coda, Alarm := #Alarm.Coda.Enc);   // "PosFbk_SickAFM60"
END_REGION

REGION Network 60: [Ax] - Axis 2 Manger
   RUNG wire#powerrail
      #Ax_Coda(AreaInterface := #AreaInterface, ZSI := #ZSI, DSI := #DSI_Feed_Coda, Drive :=, DataIn :=, CIn :=, Config := #Config.Navetta.Coda.Ax, HW_ID_TEL1 :=, PosFeedback := #Enc_Coda_ITF, Par := #Par.Ax_Man, Pers_Data := #Par.Ax_Coda_Pers, Warning := #Warning.Coda.Ax, Alarm := #Alarm.Coda.Ax, MachineInterface =>, DataOut =>, COut => #COut.Coda.Ax)
   END_RUNG
   // the same network as SCL:
   #Ax_Coda(AreaInterface := #AreaInterface,   // "Positioning_DOL_Machine_FB"
            ZSI := #ZSI,
            DSI := #DSI_Feed_Coda,
            Config := #Config.Navetta.Coda.Ax,
            PosFeedback := #Enc_Coda_ITF,
            Par := #Par.Ax_Man,
            Pers_Data := #Par.Ax_Coda_Pers,
            Warning := #Warning.Coda.Ax,
            Alarm := #Alarm.Coda.Ax,
            COut => #COut.Coda.Ax);
END_REGION

REGION Network 62: <<< PALETTI INTRENI >>>
END_REGION

REGION Network 63: Paletti Interni - CIn External alarm
   RUNG wire#powerrail
      Contact( FALSE )
      Coil( #PalettiInterni_Coda.Cin.ExternalAlarms )
   END_RUNG
   // the same network as SCL:
   #PalettiInterni_Coda.Cin.ExternalAlarms := FALSE;
END_REGION

REGION Network 64: Paletti Interni - Cin Ext Enable
   RUNG wire#powerrail
      Contact( #CIn.Manager.Control_ON )
      wire#w1
      Coil( #PalettiInterni_Coda.Cin.Rest_ExtEnable )
   END_RUNG
   RUNG wire#powerrail
      Contact( #AreaInterface.Man )
      I_Contact( #CIn.Manager.Control_ON )
      Contact( #Sts.OP_CanMoveFreely )
   END_RUNG wire#w1
   RUNG wire#powerrail
      Contact( #CIn.Manager.Control_ON )
      wire#w2
      Coil( #PalettiInterni_Coda.Cin.Work_ExtEnable )
   END_RUNG
   RUNG wire#powerrail
      Contact( #AreaInterface.Man )
      I_Contact( #CIn.Manager.Control_ON )
      Contact( #Sts.OP_CanMoveFreely )
   END_RUNG wire#w2
   // the same network as SCL:
   #PalettiInterni_Coda.Cin.Rest_ExtEnable := #CIn.Manager.Control_ON OR (#AreaInterface.Man AND NOT #CIn.Manager.Control_ON AND #Sts.OP_CanMoveFreely);
   #PalettiInterni_Coda.Cin.Work_ExtEnable := #CIn.Manager.Control_ON OR (#AreaInterface.Man AND NOT #CIn.Manager.Control_ON AND #Sts.OP_CanMoveFreely);
END_REGION

REGION Network 65: Paletti Interni - Data In
   RUNG wire#powerrail
      Contact( #DataIn.PalettoInternoCoda_LsRest )
      Coil( #PalettiInterni_Coda.DataIn.Rest_Ls[1] )
   END_RUNG
   RUNG wire#powerrail
      Contact( #DataIn.PalettoInternoCoda_LsWork )
      Coil( #PalettiInterni_Coda.DataIn.Work_Ls[1] )
   END_RUNG
   // the same network as SCL:
   #PalettiInterni_Coda.DataIn.Rest_Ls[1] := #DataIn.PalettoInternoCoda_LsRest;
   #PalettiInterni_Coda.DataIn.Work_Ls[1] := #DataIn.PalettoInternoCoda_LsWork;
END_REGION

REGION Network 66: Valve Manager
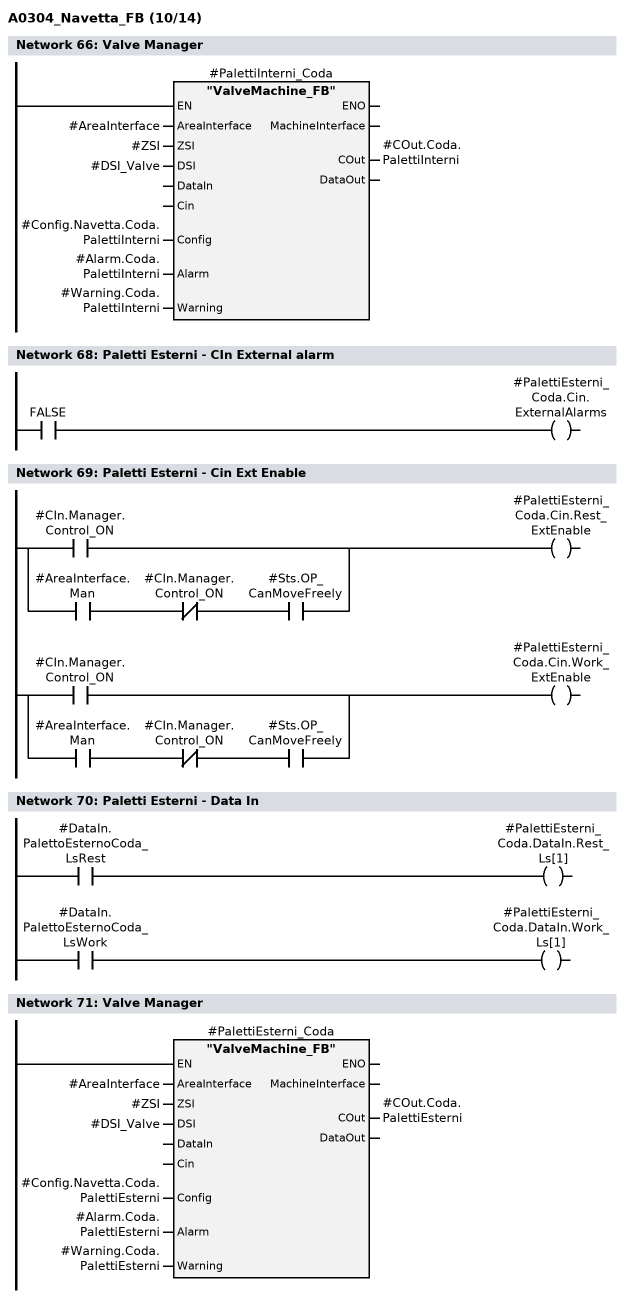
   RUNG wire#powerrail
      #PalettiInterni_Coda(AreaInterface := #AreaInterface, ZSI := #ZSI, DSI := #DSI_Valve, DataIn :=, Cin :=, Config := #Config.Navetta.Coda.PalettiInterni, Alarm := #Alarm.Coda.PalettiInterni, Warning := #Warning.Coda.PalettiInterni, MachineInterface =>, COut => #COut.Coda.PalettiInterni, DataOut =>)
   END_RUNG
   // the same network as SCL:
   #PalettiInterni_Coda(AreaInterface := #AreaInterface,   // "ValveMachine_FB"
                        ZSI := #ZSI,
                        DSI := #DSI_Valve,
                        Config := #Config.Navetta.Coda.PalettiInterni,
                        Alarm := #Alarm.Coda.PalettiInterni,
                        Warning := #Warning.Coda.PalettiInterni,
                        COut => #COut.Coda.PalettiInterni);
END_REGION

REGION Network 67: <<< PALETTI ESTERNI>>>
END_REGION

REGION Network 68: Paletti Esterni - CIn External alarm
   RUNG wire#powerrail
      Contact( FALSE )
      Coil( #PalettiEsterni_Coda.Cin.ExternalAlarms )
   END_RUNG
   // the same network as SCL:
   #PalettiEsterni_Coda.Cin.ExternalAlarms := FALSE;
END_REGION

REGION Network 69: Paletti Esterni - Cin Ext Enable
   RUNG wire#powerrail
      Contact( #CIn.Manager.Control_ON )
      wire#w1
      Coil( #PalettiEsterni_Coda.Cin.Rest_ExtEnable )
   END_RUNG
   RUNG wire#powerrail
      Contact( #AreaInterface.Man )
      I_Contact( #CIn.Manager.Control_ON )
      Contact( #Sts.OP_CanMoveFreely )
   END_RUNG wire#w1
   RUNG wire#powerrail
      Contact( #CIn.Manager.Control_ON )
      wire#w2
      Coil( #PalettiEsterni_Coda.Cin.Work_ExtEnable )
   END_RUNG
   RUNG wire#powerrail
      Contact( #AreaInterface.Man )
      I_Contact( #CIn.Manager.Control_ON )
      Contact( #Sts.OP_CanMoveFreely )
   END_RUNG wire#w2
   // the same network as SCL:
   #PalettiEsterni_Coda.Cin.Rest_ExtEnable := #CIn.Manager.Control_ON OR (#AreaInterface.Man AND NOT #CIn.Manager.Control_ON AND #Sts.OP_CanMoveFreely);
   #PalettiEsterni_Coda.Cin.Work_ExtEnable := #CIn.Manager.Control_ON OR (#AreaInterface.Man AND NOT #CIn.Manager.Control_ON AND #Sts.OP_CanMoveFreely);
END_REGION

REGION Network 70: Paletti Esterni - Data In
   RUNG wire#powerrail
      Contact( #DataIn.PalettoEsternoCoda_LsRest )
      Coil( #PalettiEsterni_Coda.DataIn.Rest_Ls[1] )
   END_RUNG
   RUNG wire#powerrail
      Contact( #DataIn.PalettoEsternoCoda_LsWork )
      Coil( #PalettiEsterni_Coda.DataIn.Work_Ls[1] )
   END_RUNG
   // the same network as SCL:
   #PalettiEsterni_Coda.DataIn.Rest_Ls[1] := #DataIn.PalettoEsternoCoda_LsRest;
   #PalettiEsterni_Coda.DataIn.Work_Ls[1] := #DataIn.PalettoEsternoCoda_LsWork;
END_REGION

REGION Network 71: Valve Manager
   RUNG wire#powerrail
      #PalettiEsterni_Coda(AreaInterface := #AreaInterface, ZSI := #ZSI, DSI := #DSI_Valve, DataIn :=, Cin :=, Config := #Config.Navetta.Coda.PalettiEsterni, Alarm := #Alarm.Coda.PalettiEsterni, Warning := #Warning.Coda.PalettiEsterni, MachineInterface =>, COut => #COut.Coda.PalettiEsterni, DataOut =>)
   END_RUNG
   // the same network as SCL:
   #PalettiEsterni_Coda(AreaInterface := #AreaInterface,   // "ValveMachine_FB"
                        ZSI := #ZSI,
                        DSI := #DSI_Valve,
                        Config := #Config.Navetta.Coda.PalettiEsterni,
                        Alarm := #Alarm.Coda.PalettiEsterni,
                        Warning := #Warning.Coda.PalettiEsterni,
                        COut => #COut.Coda.PalettiEsterni);
END_REGION

REGION Network 73: Request Reload Air
   // Serve perche al primo comando dopo che viene a mancare l'aria il cilindro uscirebbe troppo velocemente quindi vengono riempite le due camera d'aria del cilindro con il blocco stelo inserito in modo da riempirle senza muovere nulla
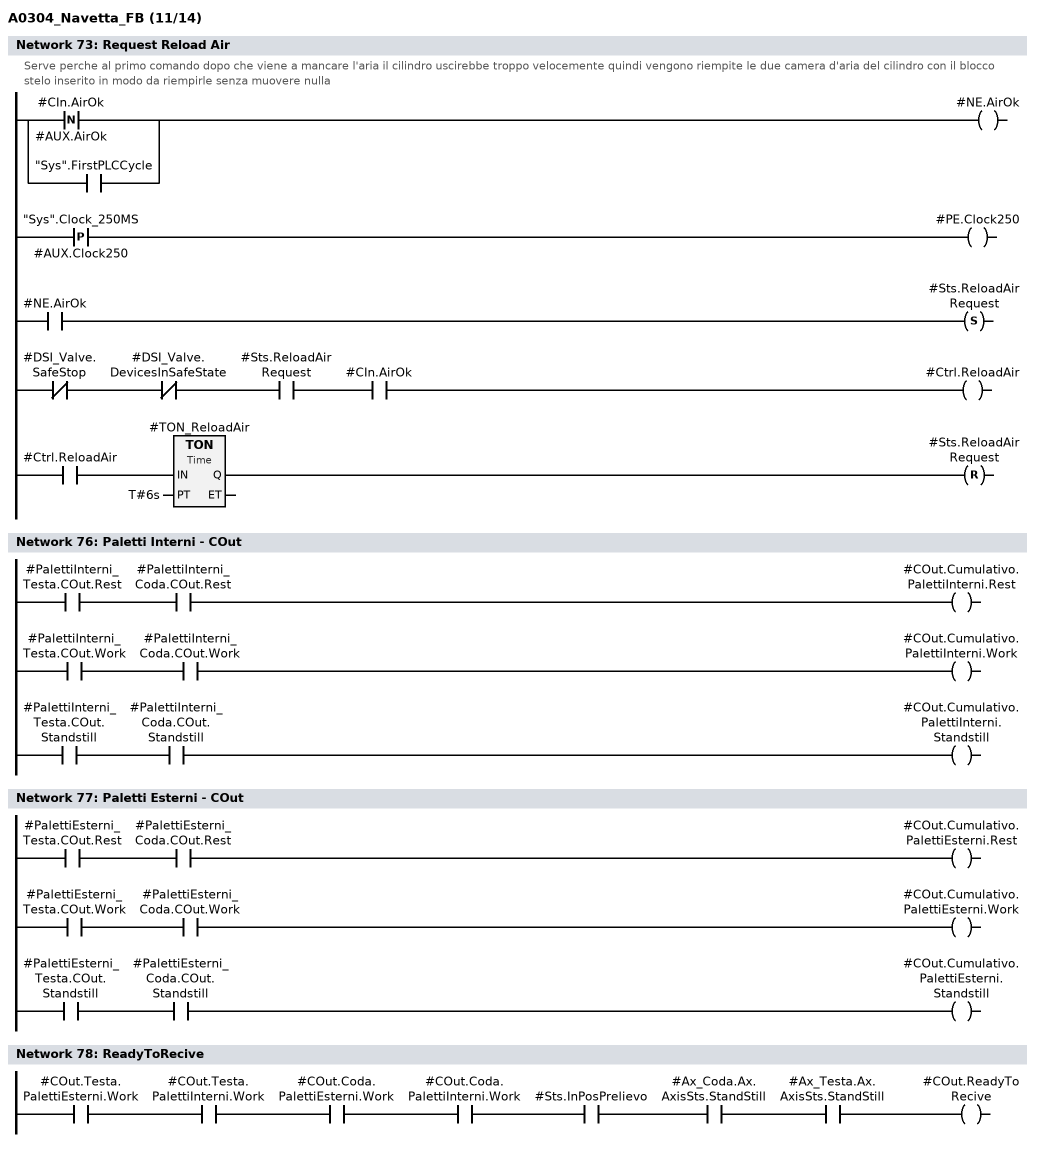
   RUNG wire#powerrail
      N_Contact(operand := #CIn.AirOk, bit := #AUX.AirOk)
      wire#w1
      Coil( #NE.AirOk )
   END_RUNG
   RUNG wire#powerrail
      Contact( "Sys".FirstPLCCycle )
   END_RUNG wire#w1
   RUNG wire#powerrail
      P_Contact(operand := "Sys".Clock_250MS, bit := #AUX.Clock250)
      Coil( #PE.Clock250 )
   END_RUNG
   RUNG wire#powerrail
      Contact( #NE.AirOk )
      S_Coil( #Sts.ReloadAirRequest )
   END_RUNG
   RUNG wire#powerrail
      I_Contact( #DSI_Valve.SafeStop )
      I_Contact( #DSI_Valve.DevicesInSafeState )
      Contact( #Sts.ReloadAirRequest )
      Contact( #CIn.AirOk )
      Coil( #Ctrl.ReloadAir )
   END_RUNG
   RUNG wire#powerrail
      Contact( #Ctrl.ReloadAir )
      { S7_Templates := "time_type := Time" } #TON_ReloadAir.TON(pt := T#6s, et =>)
      R_Coil( #Sts.ReloadAirRequest )
   END_RUNG
   // the same network as SCL:
   #_w1 := NOT #CIn.AirOk AND #AUX.AirOk;   // falling edge of #CIn.AirOk
   #AUX.AirOk := #CIn.AirOk;
   #NE.AirOk := #_w1 OR "Sys".FirstPLCCycle;
   #_w2 := "Sys".Clock_250MS AND NOT #AUX.Clock250;   // rising edge of "Sys".Clock_250MS
   #AUX.Clock250 := "Sys".Clock_250MS;
   #PE.Clock250 := #_w2;
   IF #NE.AirOk THEN #Sts.ReloadAirRequest := TRUE; END_IF;
   #Ctrl.ReloadAir := NOT #DSI_Valve.SafeStop AND NOT #DSI_Valve.DevicesInSafeState AND #Sts.ReloadAirRequest AND #CIn.AirOk;
   #TON_ReloadAir.TON(IN := #Ctrl.ReloadAir, PT := T#6s);
   IF #TON_ReloadAir.Q THEN #Sts.ReloadAirRequest := FALSE; END_IF;
END_REGION

REGION Network 75: <<< COut >>>
END_REGION

REGION Network 76: Paletti Interni - COut
   RUNG wire#powerrail
      Contact( #PalettiInterni_Testa.COut.Rest )
      Contact( #PalettiInterni_Coda.COut.Rest )
      Coil( #COut.Cumulativo.PalettiInterni.Rest )
   END_RUNG
   RUNG wire#powerrail
      Contact( #PalettiInterni_Testa.COut.Work )
      Contact( #PalettiInterni_Coda.COut.Work )
      Coil( #COut.Cumulativo.PalettiInterni.Work )
   END_RUNG
   RUNG wire#powerrail
      Contact( #PalettiInterni_Testa.COut.Standstill )
      Contact( #PalettiInterni_Coda.COut.Standstill )
      Coil( #COut.Cumulativo.PalettiInterni.Standstill )
   END_RUNG
   // the same network as SCL:
   #COut.Cumulativo.PalettiInterni.Rest := #PalettiInterni_Testa.COut.Rest AND #PalettiInterni_Coda.COut.Rest;
   #COut.Cumulativo.PalettiInterni.Work := #PalettiInterni_Testa.COut.Work AND #PalettiInterni_Coda.COut.Work;
   #COut.Cumulativo.PalettiInterni.Standstill := #PalettiInterni_Testa.COut.Standstill AND #PalettiInterni_Coda.COut.Standstill;
END_REGION

REGION Network 77: Paletti Esterni - COut
   RUNG wire#powerrail
      Contact( #PalettiEsterni_Testa.COut.Rest )
      Contact( #PalettiEsterni_Coda.COut.Rest )
      Coil( #COut.Cumulativo.PalettiEsterni.Rest )
   END_RUNG
   RUNG wire#powerrail
      Contact( #PalettiEsterni_Testa.COut.Work )
      Contact( #PalettiEsterni_Coda.COut.Work )
      Coil( #COut.Cumulativo.PalettiEsterni.Work )
   END_RUNG
   RUNG wire#powerrail
      Contact( #PalettiEsterni_Testa.COut.Standstill )
      Contact( #PalettiEsterni_Coda.COut.Standstill )
      Coil( #COut.Cumulativo.PalettiEsterni.Standstill )
   END_RUNG
   // the same network as SCL:
   #COut.Cumulativo.PalettiEsterni.Rest := #PalettiEsterni_Testa.COut.Rest AND #PalettiEsterni_Coda.COut.Rest;
   #COut.Cumulativo.PalettiEsterni.Work := #PalettiEsterni_Testa.COut.Work AND #PalettiEsterni_Coda.COut.Work;
   #COut.Cumulativo.PalettiEsterni.Standstill := #PalettiEsterni_Testa.COut.Standstill AND #PalettiEsterni_Coda.COut.Standstill;
END_REGION

REGION Network 78: ReadyToRecive
   RUNG wire#powerrail
      Contact( #COut.Testa.PalettiEsterni.Work )
      Contact( #COut.Testa.PalettiInterni.Work )
      Contact( #COut.Coda.PalettiEsterni.Work )
      Contact( #COut.Coda.PalettiInterni.Work )
      Contact( #Sts.InPosPrelievo )
      Contact( #Ax_Coda.Ax.AxisSts.StandStill )
      Contact( #Ax_Testa.Ax.AxisSts.StandStill )
      Coil( #COut.ReadyToRecive )
   END_RUNG
   // the same network as SCL:
   #COut.ReadyToRecive := #COut.Testa.PalettiEsterni.Work AND #COut.Testa.PalettiInterni.Work AND #COut.Coda.PalettiEsterni.Work AND #COut.Coda.PalettiInterni.Work AND #Sts.InPosPrelievo AND #Ax_Coda.Ax.AxisSts.StandStill AND #Ax_Testa.Ax.AxisSts.StandStill;
END_REGION

REGION Network 80: <<< DataOut >>>
END_REGION

REGION Network 81: Paletto Esterno- Testa
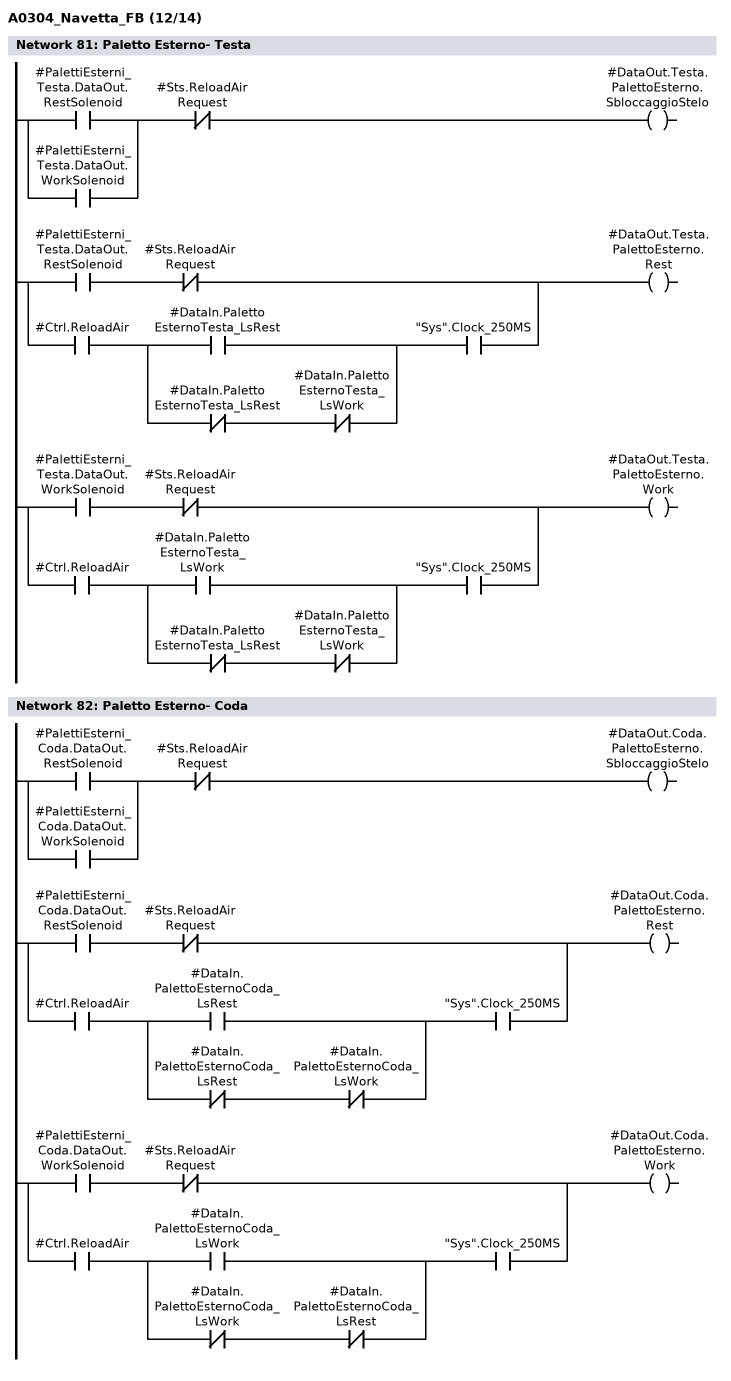
   RUNG wire#powerrail
      Contact( #PalettiEsterni_Testa.DataOut.RestSolenoid )
      wire#w1
      I_Contact( #Sts.ReloadAirRequest )
      Coil( #DataOut.Testa.PalettoEsterno.SbloccaggioStelo )
   END_RUNG
   RUNG wire#powerrail
      Contact( #PalettiEsterni_Testa.DataOut.WorkSolenoid )
   END_RUNG wire#w1
   RUNG wire#powerrail
      Contact( #PalettiEsterni_Testa.DataOut.RestSolenoid )
      I_Contact( #Sts.ReloadAirRequest )
      wire#w2
      Coil( #DataOut.Testa.PalettoEsterno.Rest )
   END_RUNG
   RUNG wire#powerrail
      Contact( #Ctrl.ReloadAir )
      wire#w3
      Contact( #DataIn.PalettoEsternoTesta_LsRest )
      wire#w4
      Contact( "Sys".Clock_250MS )
   END_RUNG wire#w2
   RUNG wire#w3
      I_Contact( #DataIn.PalettoEsternoTesta_LsRest )
      I_Contact( #DataIn.PalettoEsternoTesta_LsWork )
   END_RUNG wire#w4
   RUNG wire#powerrail
      Contact( #PalettiEsterni_Testa.DataOut.WorkSolenoid )
      I_Contact( #Sts.ReloadAirRequest )
      wire#w5
      Coil( #DataOut.Testa.PalettoEsterno.Work )
   END_RUNG
   RUNG wire#powerrail
      Contact( #Ctrl.ReloadAir )
      wire#w6
      Contact( #DataIn.PalettoEsternoTesta_LsWork )
      wire#w7
      Contact( "Sys".Clock_250MS )
   END_RUNG wire#w5
   RUNG wire#w6
      I_Contact( #DataIn.PalettoEsternoTesta_LsRest )
      I_Contact( #DataIn.PalettoEsternoTesta_LsWork )
   END_RUNG wire#w7
   // the same network as SCL:
   #DataOut.Testa.PalettoEsterno.SbloccaggioStelo := (#PalettiEsterni_Testa.DataOut.RestSolenoid OR #PalettiEsterni_Testa.DataOut.WorkSolenoid) AND NOT #Sts.ReloadAirRequest;
   #DataOut.Testa.PalettoEsterno.Rest := (#PalettiEsterni_Testa.DataOut.RestSolenoid AND NOT #Sts.ReloadAirRequest) OR (#Ctrl.ReloadAir AND (#DataIn.PalettoEsternoTesta_LsRest OR (NOT #DataIn.PalettoEsternoTesta_LsRest AND NOT #DataIn.PalettoEsternoTesta_LsWork)) AND "Sys".Clock_250MS);
   #DataOut.Testa.PalettoEsterno.Work := (#PalettiEsterni_Testa.DataOut.WorkSolenoid AND NOT #Sts.ReloadAirRequest) OR (#Ctrl.ReloadAir AND (#DataIn.PalettoEsternoTesta_LsWork OR (NOT #DataIn.PalettoEsternoTesta_LsRest AND NOT #DataIn.PalettoEsternoTesta_LsWork)) AND "Sys".Clock_250MS);
END_REGION

REGION Network 82: Paletto Esterno- Coda
   RUNG wire#powerrail
      Contact( #PalettiEsterni_Coda.DataOut.RestSolenoid )
      wire#w1
      I_Contact( #Sts.ReloadAirRequest )
      Coil( #DataOut.Coda.PalettoEsterno.SbloccaggioStelo )
   END_RUNG
   RUNG wire#powerrail
      Contact( #PalettiEsterni_Coda.DataOut.WorkSolenoid )
   END_RUNG wire#w1
   RUNG wire#powerrail
      Contact( #PalettiEsterni_Coda.DataOut.RestSolenoid )
      I_Contact( #Sts.ReloadAirRequest )
      wire#w2
      Coil( #DataOut.Coda.PalettoEsterno.Rest )
   END_RUNG
   RUNG wire#powerrail
      Contact( #Ctrl.ReloadAir )
      wire#w3
      Contact( #DataIn.PalettoEsternoCoda_LsRest )
      wire#w4
      Contact( "Sys".Clock_250MS )
   END_RUNG wire#w2
   RUNG wire#w3
      I_Contact( #DataIn.PalettoEsternoCoda_LsRest )
      I_Contact( #DataIn.PalettoEsternoCoda_LsWork )
   END_RUNG wire#w4
   RUNG wire#powerrail
      Contact( #PalettiEsterni_Coda.DataOut.WorkSolenoid )
      I_Contact( #Sts.ReloadAirRequest )
      wire#w5
      Coil( #DataOut.Coda.PalettoEsterno.Work )
   END_RUNG
   RUNG wire#powerrail
      Contact( #Ctrl.ReloadAir )
      wire#w6
      Contact( #DataIn.PalettoEsternoCoda_LsWork )
      wire#w7
      Contact( "Sys".Clock_250MS )
   END_RUNG wire#w5
   RUNG wire#w6
      I_Contact( #DataIn.PalettoEsternoCoda_LsWork )
      I_Contact( #DataIn.PalettoEsternoCoda_LsRest )
   END_RUNG wire#w7
   // the same network as SCL:
   #DataOut.Coda.PalettoEsterno.SbloccaggioStelo := (#PalettiEsterni_Coda.DataOut.RestSolenoid OR #PalettiEsterni_Coda.DataOut.WorkSolenoid) AND NOT #Sts.ReloadAirRequest;
   #DataOut.Coda.PalettoEsterno.Rest := (#PalettiEsterni_Coda.DataOut.RestSolenoid AND NOT #Sts.ReloadAirRequest) OR (#Ctrl.ReloadAir AND (#DataIn.PalettoEsternoCoda_LsRest OR (NOT #DataIn.PalettoEsternoCoda_LsRest AND NOT #DataIn.PalettoEsternoCoda_LsWork)) AND "Sys".Clock_250MS);
   #DataOut.Coda.PalettoEsterno.Work := (#PalettiEsterni_Coda.DataOut.WorkSolenoid AND NOT #Sts.ReloadAirRequest) OR (#Ctrl.ReloadAir AND (#DataIn.PalettoEsternoCoda_LsWork OR (NOT #DataIn.PalettoEsternoCoda_LsWork AND NOT #DataIn.PalettoEsternoCoda_LsRest)) AND "Sys".Clock_250MS);
END_REGION

REGION Network 83: Paletto Interno- Testa
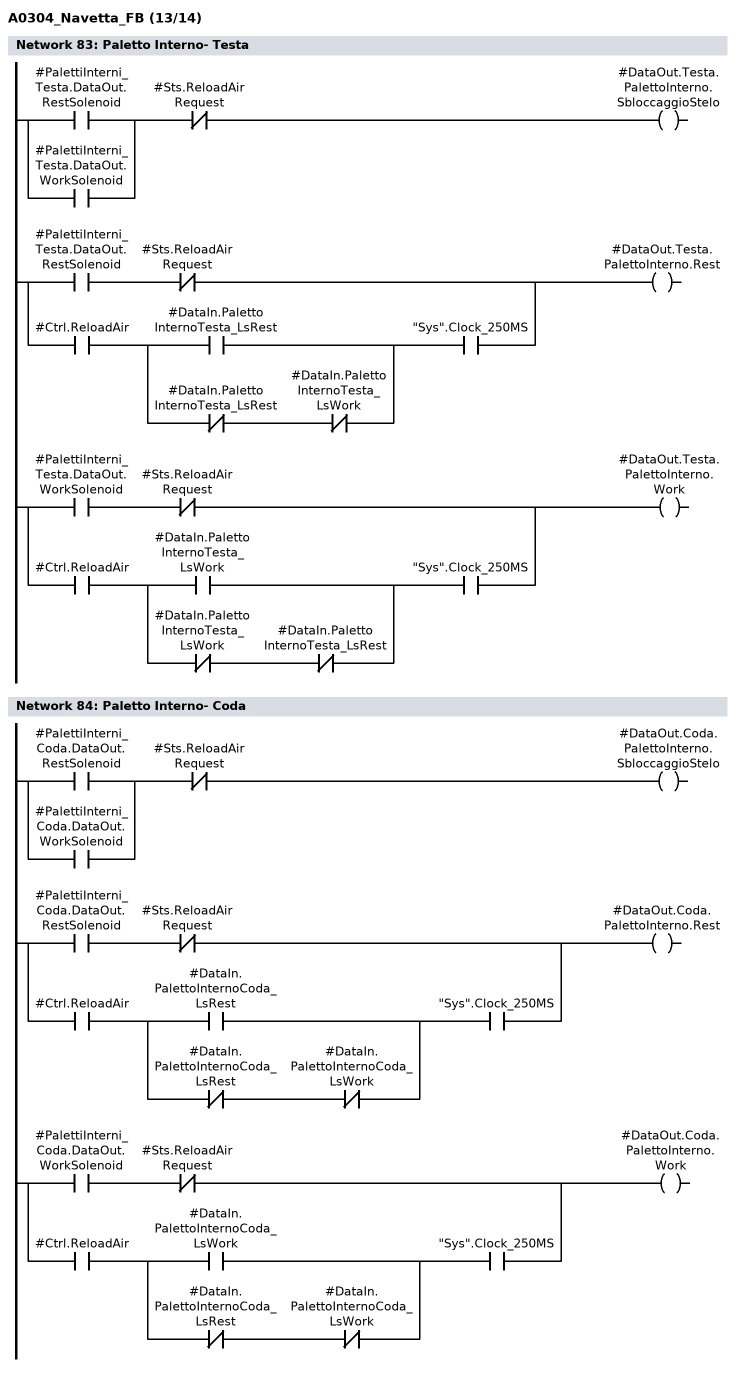
   RUNG wire#powerrail
      Contact( #PalettiInterni_Testa.DataOut.RestSolenoid )
      wire#w1
      I_Contact( #Sts.ReloadAirRequest )
      Coil( #DataOut.Testa.PalettoInterno.SbloccaggioStelo )
   END_RUNG
   RUNG wire#powerrail
      Contact( #PalettiInterni_Testa.DataOut.WorkSolenoid )
   END_RUNG wire#w1
   RUNG wire#powerrail
      Contact( #PalettiInterni_Testa.DataOut.RestSolenoid )
      I_Contact( #Sts.ReloadAirRequest )
      wire#w2
      Coil( #DataOut.Testa.PalettoInterno.Rest )
   END_RUNG
   RUNG wire#powerrail
      Contact( #Ctrl.ReloadAir )
      wire#w3
      Contact( #DataIn.PalettoInternoTesta_LsRest )
      wire#w4
      Contact( "Sys".Clock_250MS )
   END_RUNG wire#w2
   RUNG wire#w3
      I_Contact( #DataIn.PalettoInternoTesta_LsRest )
      I_Contact( #DataIn.PalettoInternoTesta_LsWork )
   END_RUNG wire#w4
   RUNG wire#powerrail
      Contact( #PalettiInterni_Testa.DataOut.WorkSolenoid )
      I_Contact( #Sts.ReloadAirRequest )
      wire#w5
      Coil( #DataOut.Testa.PalettoInterno.Work )
   END_RUNG
   RUNG wire#powerrail
      Contact( #Ctrl.ReloadAir )
      wire#w6
      Contact( #DataIn.PalettoInternoTesta_LsWork )
      wire#w7
      Contact( "Sys".Clock_250MS )
   END_RUNG wire#w5
   RUNG wire#w6
      I_Contact( #DataIn.PalettoInternoTesta_LsWork )
      I_Contact( #DataIn.PalettoInternoTesta_LsRest )
   END_RUNG wire#w7
   // the same network as SCL:
   #DataOut.Testa.PalettoInterno.SbloccaggioStelo := (#PalettiInterni_Testa.DataOut.RestSolenoid OR #PalettiInterni_Testa.DataOut.WorkSolenoid) AND NOT #Sts.ReloadAirRequest;
   #DataOut.Testa.PalettoInterno.Rest := (#PalettiInterni_Testa.DataOut.RestSolenoid AND NOT #Sts.ReloadAirRequest) OR (#Ctrl.ReloadAir AND (#DataIn.PalettoInternoTesta_LsRest OR (NOT #DataIn.PalettoInternoTesta_LsRest AND NOT #DataIn.PalettoInternoTesta_LsWork)) AND "Sys".Clock_250MS);
   #DataOut.Testa.PalettoInterno.Work := (#PalettiInterni_Testa.DataOut.WorkSolenoid AND NOT #Sts.ReloadAirRequest) OR (#Ctrl.ReloadAir AND (#DataIn.PalettoInternoTesta_LsWork OR (NOT #DataIn.PalettoInternoTesta_LsWork AND NOT #DataIn.PalettoInternoTesta_LsRest)) AND "Sys".Clock_250MS);
END_REGION

REGION Network 84: Paletto Interno- Coda
   RUNG wire#powerrail
      Contact( #PalettiInterni_Coda.DataOut.RestSolenoid )
      wire#w1
      I_Contact( #Sts.ReloadAirRequest )
      Coil( #DataOut.Coda.PalettoInterno.SbloccaggioStelo )
   END_RUNG
   RUNG wire#powerrail
      Contact( #PalettiInterni_Coda.DataOut.WorkSolenoid )
   END_RUNG wire#w1
   RUNG wire#powerrail
      Contact( #PalettiInterni_Coda.DataOut.RestSolenoid )
      I_Contact( #Sts.ReloadAirRequest )
      wire#w2
      Coil( #DataOut.Coda.PalettoInterno.Rest )
   END_RUNG
   RUNG wire#powerrail
      Contact( #Ctrl.ReloadAir )
      wire#w3
      Contact( #DataIn.PalettoInternoCoda_LsRest )
      wire#w4
      Contact( "Sys".Clock_250MS )
   END_RUNG wire#w2
   RUNG wire#w3
      I_Contact( #DataIn.PalettoInternoCoda_LsRest )
      I_Contact( #DataIn.PalettoInternoCoda_LsWork )
   END_RUNG wire#w4
   RUNG wire#powerrail
      Contact( #PalettiInterni_Coda.DataOut.WorkSolenoid )
      I_Contact( #Sts.ReloadAirRequest )
      wire#w5
      Coil( #DataOut.Coda.PalettoInterno.Work )
   END_RUNG
   RUNG wire#powerrail
      Contact( #Ctrl.ReloadAir )
      wire#w6
      Contact( #DataIn.PalettoInternoCoda_LsWork )
      wire#w7
      Contact( "Sys".Clock_250MS )
   END_RUNG wire#w5
   RUNG wire#w6
      I_Contact( #DataIn.PalettoInternoCoda_LsRest )
      I_Contact( #DataIn.PalettoInternoCoda_LsWork )
   END_RUNG wire#w7
   // the same network as SCL:
   #DataOut.Coda.PalettoInterno.SbloccaggioStelo := (#PalettiInterni_Coda.DataOut.RestSolenoid OR #PalettiInterni_Coda.DataOut.WorkSolenoid) AND NOT #Sts.ReloadAirRequest;
   #DataOut.Coda.PalettoInterno.Rest := (#PalettiInterni_Coda.DataOut.RestSolenoid AND NOT #Sts.ReloadAirRequest) OR (#Ctrl.ReloadAir AND (#DataIn.PalettoInternoCoda_LsRest OR (NOT #DataIn.PalettoInternoCoda_LsRest AND NOT #DataIn.PalettoInternoCoda_LsWork)) AND "Sys".Clock_250MS);
   #DataOut.Coda.PalettoInterno.Work := (#PalettiInterni_Coda.DataOut.WorkSolenoid AND NOT #Sts.ReloadAirRequest) OR (#Ctrl.ReloadAir AND (#DataIn.PalettoInternoCoda_LsWork OR (NOT #DataIn.PalettoInternoCoda_LsRest AND NOT #DataIn.PalettoInternoCoda_LsWork)) AND "Sys".Clock_250MS);
END_REGION

REGION Network 86: <<< MACHINE STATUS >>>
END_REGION

REGION Network 87: Collect machine to zone interface (internal machines OR)
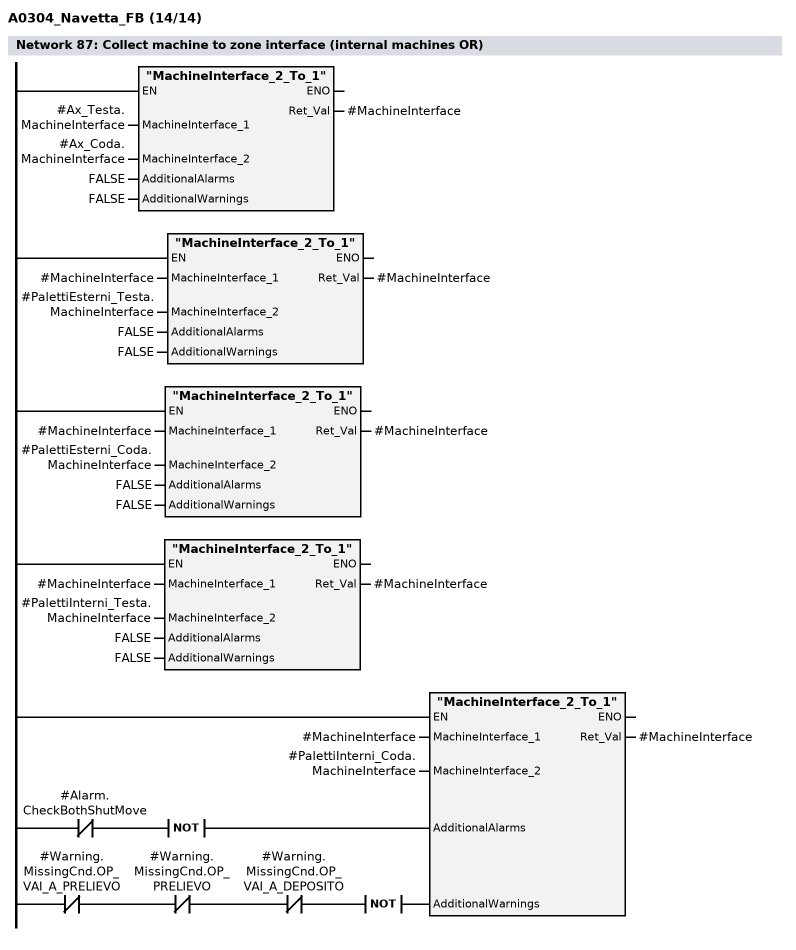
   RUNG wire#powerrail
      "MachineInterface_2_To_1"(MachineInterface_1 := #Ax_Testa.MachineInterface, MachineInterface_2 := #Ax_Coda.MachineInterface, AdditionalAlarms := FALSE, AdditionalWarnings := FALSE, Ret_Val => #MachineInterface)
   END_RUNG
   RUNG wire#powerrail
      "MachineInterface_2_To_1"(MachineInterface_1 := #MachineInterface, MachineInterface_2 := #PalettiEsterni_Testa.MachineInterface, AdditionalAlarms := FALSE, AdditionalWarnings := FALSE, Ret_Val => #MachineInterface)
   END_RUNG
   RUNG wire#powerrail
      "MachineInterface_2_To_1"(MachineInterface_1 := #MachineInterface, MachineInterface_2 := #PalettiEsterni_Coda.MachineInterface, AdditionalAlarms := FALSE, AdditionalWarnings := FALSE, Ret_Val => #MachineInterface)
   END_RUNG
   RUNG wire#powerrail
      "MachineInterface_2_To_1"(MachineInterface_1 := #MachineInterface, MachineInterface_2 := #PalettiInterni_Testa.MachineInterface, AdditionalAlarms := FALSE, AdditionalWarnings := FALSE, Ret_Val => #MachineInterface)
   END_RUNG
   RUNG wire#powerrail
      "MachineInterface_2_To_1"(AdditionalAlarms := wire#w1, AdditionalWarnings := wire#w2, MachineInterface_1 := #MachineInterface, MachineInterface_2 := #PalettiInterni_Coda.MachineInterface, Ret_Val => #MachineInterface)
   END_RUNG
   RUNG wire#powerrail
      I_Contact( #Alarm.CheckBothShutMove )
      Not()
   END_RUNG wire#w1
   RUNG wire#powerrail
      I_Contact( #Warning.MissingCnd.OP_VAI_A_PRELIEVO )
      I_Contact( #Warning.MissingCnd.OP_PRELIEVO )
      I_Contact( #Warning.MissingCnd.OP_VAI_A_DEPOSITO )
      Not()
   END_RUNG wire#w2
   // the same network as SCL:
   #MachineInterface := "MachineInterface_2_To_1"(MachineInterface_1 := #Ax_Testa.MachineInterface,
                           MachineInterface_2 := #Ax_Coda.MachineInterface,
                           AdditionalAlarms := FALSE,
                           AdditionalWarnings := FALSE);
   #MachineInterface := "MachineInterface_2_To_1"(MachineInterface_1 := #MachineInterface,
                           MachineInterface_2 := #PalettiEsterni_Testa.MachineInterface,
                           AdditionalAlarms := FALSE,
                           AdditionalWarnings := FALSE);
   #MachineInterface := "MachineInterface_2_To_1"(MachineInterface_1 := #MachineInterface,
                           MachineInterface_2 := #PalettiEsterni_Coda.MachineInterface,
                           AdditionalAlarms := FALSE,
                           AdditionalWarnings := FALSE);
   #MachineInterface := "MachineInterface_2_To_1"(MachineInterface_1 := #MachineInterface,
                           MachineInterface_2 := #PalettiInterni_Testa.MachineInterface,
                           AdditionalAlarms := FALSE,
                           AdditionalWarnings := FALSE);
   #MachineInterface := "MachineInterface_2_To_1"(MachineInterface_1 := #MachineInterface,
                           MachineInterface_2 := #PalettiInterni_Coda.MachineInterface,
                           AdditionalAlarms := NOT (NOT #Alarm.CheckBothShutMove),
                           AdditionalWarnings := NOT (NOT #Warning.MissingCnd.OP_VAI_A_PRELIEVO AND NOT #Warning.MissingCnd.OP_PRELIEVO AND NOT #Warning.MissingCnd.OP_VAI_A_DEPOSITO));
END_REGION
END_FUNCTION_BLOCK
